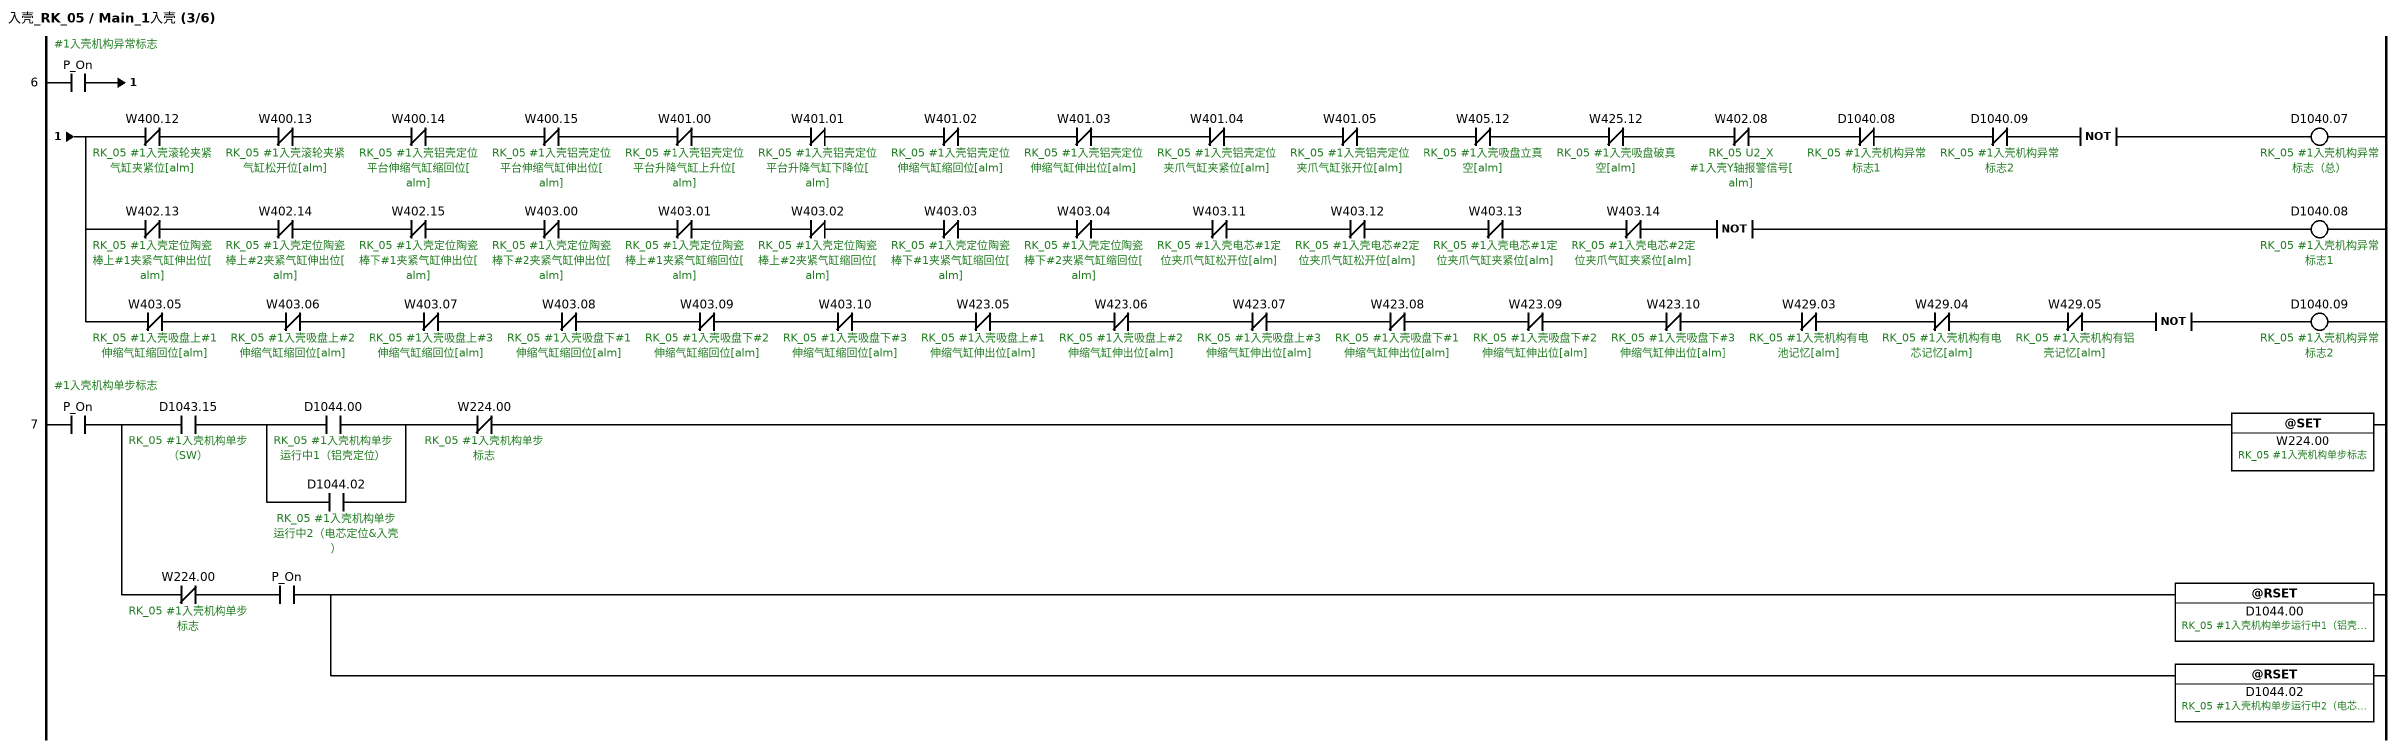
; [picture p408: 入壳_RK_05 / Main_1入壳, rungs 6-7]
; rung 6: #1入壳机构异常标志
LD P_On
OUT TR0
ANDNOT W400.12  ; RK_05 #1入壳滚轮夹紧气缸夹紧位[alm]
ANDNOT W400.13  ; RK_05 #1入壳滚轮夹紧气缸松开位[alm]
ANDNOT W400.14  ; RK_05 #1入壳铝壳定位平台伸缩气缸缩回位[alm]
ANDNOT W400.15  ; RK_05 #1入壳铝壳定位平台伸缩气缸伸出位[alm]
ANDNOT W401.00  ; RK_05 #1入壳铝壳定位平台升降气缸上升位[alm]
ANDNOT W401.01  ; RK_05 #1入壳铝壳定位平台升降气缸下降位[alm]
ANDNOT W401.02  ; RK_05 #1入壳铝壳定位伸缩气缸缩回位[alm]
ANDNOT W401.03  ; RK_05 #1入壳铝壳定位伸缩气缸伸出位[alm]
ANDNOT W401.04  ; RK_05 #1入壳铝壳定位夹爪气缸夹紧位[alm]
ANDNOT W401.05  ; RK_05 #1入壳铝壳定位夹爪气缸张开位[alm]
ANDNOT W405.12  ; RK_05 #1入壳吸盘立真空[alm]
ANDNOT W425.12  ; RK_05 #1入壳吸盘破真空[alm]
ANDNOT W402.08  ; RK_05 U2_X #1入壳Y轴报警信号[alm]
ANDNOT D1040.08  ; RK_05 #1入壳机构异常标志1
ANDNOT D1040.09  ; RK_05 #1入壳机构异常标志2
NOT(520)
OUT D1040.07  ; RK_05 #1入壳机构异常标志（总）
LD TR0
ANDNOT W402.13  ; RK_05 #1入壳定位陶瓷棒上#1夹紧气缸伸出位[alm]
ANDNOT W402.14  ; RK_05 #1入壳定位陶瓷棒上#2夹紧气缸伸出位[alm]
ANDNOT W402.15  ; RK_05 #1入壳定位陶瓷棒下#1夹紧气缸伸出位[alm]
ANDNOT W403.00  ; RK_05 #1入壳定位陶瓷棒下#2夹紧气缸伸出位[alm]
ANDNOT W403.01  ; RK_05 #1入壳定位陶瓷棒上#1夹紧气缸缩回位[alm]
ANDNOT W403.02  ; RK_05 #1入壳定位陶瓷棒上#2夹紧气缸缩回位[alm]
ANDNOT W403.03  ; RK_05 #1入壳定位陶瓷棒下#1夹紧气缸缩回位[alm]
ANDNOT W403.04  ; RK_05 #1入壳定位陶瓷棒下#2夹紧气缸缩回位[alm]
ANDNOT W403.11  ; RK_05 #1入壳电芯#1定位夹爪气缸松开位[alm]
ANDNOT W403.12  ; RK_05 #1入壳电芯#2定位夹爪气缸松开位[alm]
ANDNOT W403.13  ; RK_05 #1入壳电芯#1定位夹爪气缸夹紧位[alm]
ANDNOT W403.14  ; RK_05 #1入壳电芯#2定位夹爪气缸夹紧位[alm]
NOT(520)
OUT D1040.08  ; RK_05 #1入壳机构异常标志1
LD TR0
ANDNOT W403.05  ; RK_05 #1入壳吸盘上#1伸缩气缸缩回位[alm]
ANDNOT W403.06  ; RK_05 #1入壳吸盘上#2伸缩气缸缩回位[alm]
ANDNOT W403.07  ; RK_05 #1入壳吸盘上#3伸缩气缸缩回位[alm]
ANDNOT W403.08  ; RK_05 #1入壳吸盘下#1伸缩气缸缩回位[alm]
ANDNOT W403.09  ; RK_05 #1入壳吸盘下#2伸缩气缸缩回位[alm]
ANDNOT W403.10  ; RK_05 #1入壳吸盘下#3伸缩气缸缩回位[alm]
ANDNOT W423.05  ; RK_05 #1入壳吸盘上#1伸缩气缸伸出位[alm]
ANDNOT W423.06  ; RK_05 #1入壳吸盘上#2伸缩气缸伸出位[alm]
ANDNOT W423.07  ; RK_05 #1入壳吸盘上#3伸缩气缸伸出位[alm]
ANDNOT W423.08  ; RK_05 #1入壳吸盘下#1伸缩气缸伸出位[alm]
ANDNOT W423.09  ; RK_05 #1入壳吸盘下#2伸缩气缸伸出位[alm]
ANDNOT W423.10  ; RK_05 #1入壳吸盘下#3伸缩气缸伸出位[alm]
ANDNOT W429.03  ; RK_05 #1入壳机构有电池记忆[alm]
ANDNOT W429.04  ; RK_05 #1入壳机构有电芯记忆[alm]
ANDNOT W429.05  ; RK_05 #1入壳机构有铝壳记忆[alm]
NOT(520)
OUT D1040.09  ; RK_05 #1入壳机构异常标志2
; rung 7: #1入壳机构单步标志
LD P_On
OUT TR0
AND D1043.15  ; RK_05 #1入壳机构单步（SW）
LD D1044.00  ; RK_05 #1入壳机构单步运行中1（铝壳定位）
OR D1044.02  ; RK_05 #1入壳机构单步运行中2（电芯定位&入壳）
ANDLD
ANDNOT W224.00  ; RK_05 #1入壳机构单步标志
@SET W224.00  ; RK_05 #1入壳机构单步标志
LD TR0
ANDNOT W224.00  ; RK_05 #1入壳机构单步标志
AND P_On
@RSET D1044.00  ; RK_05 #1入壳机构单步运行中1（铝壳定位）
@RSET D1044.02  ; RK_05 #1入壳机构单步运行中2（电芯定位&入壳）

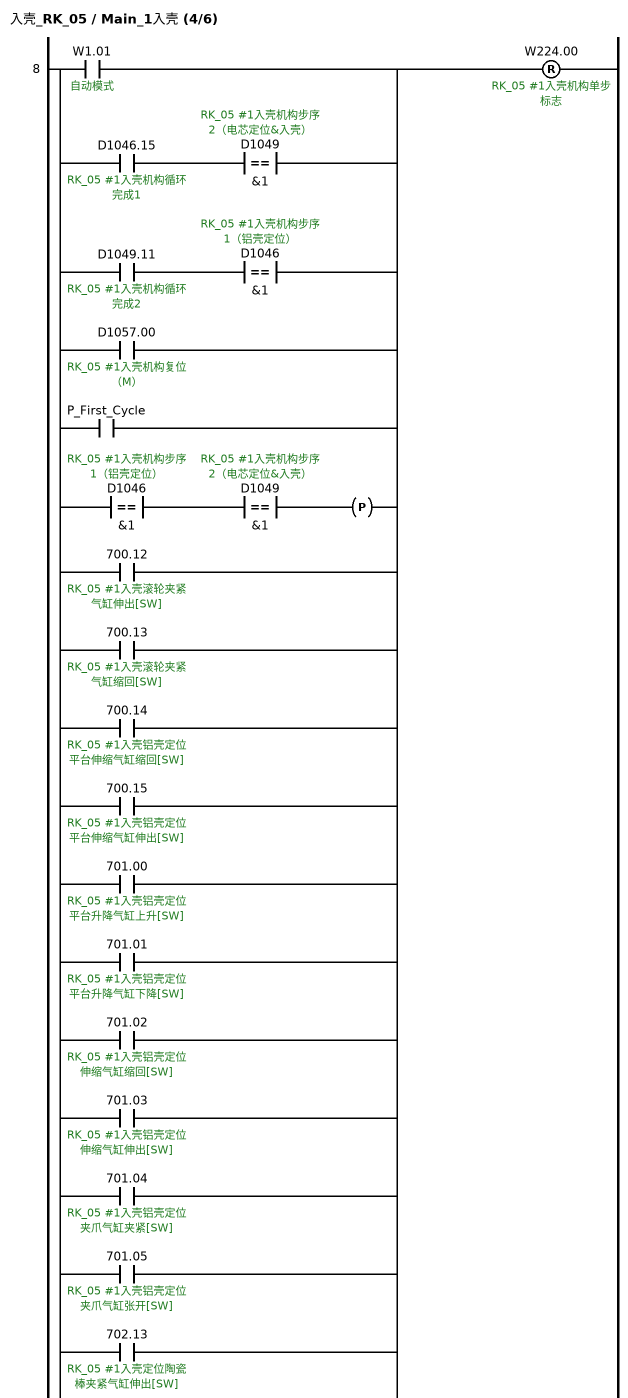

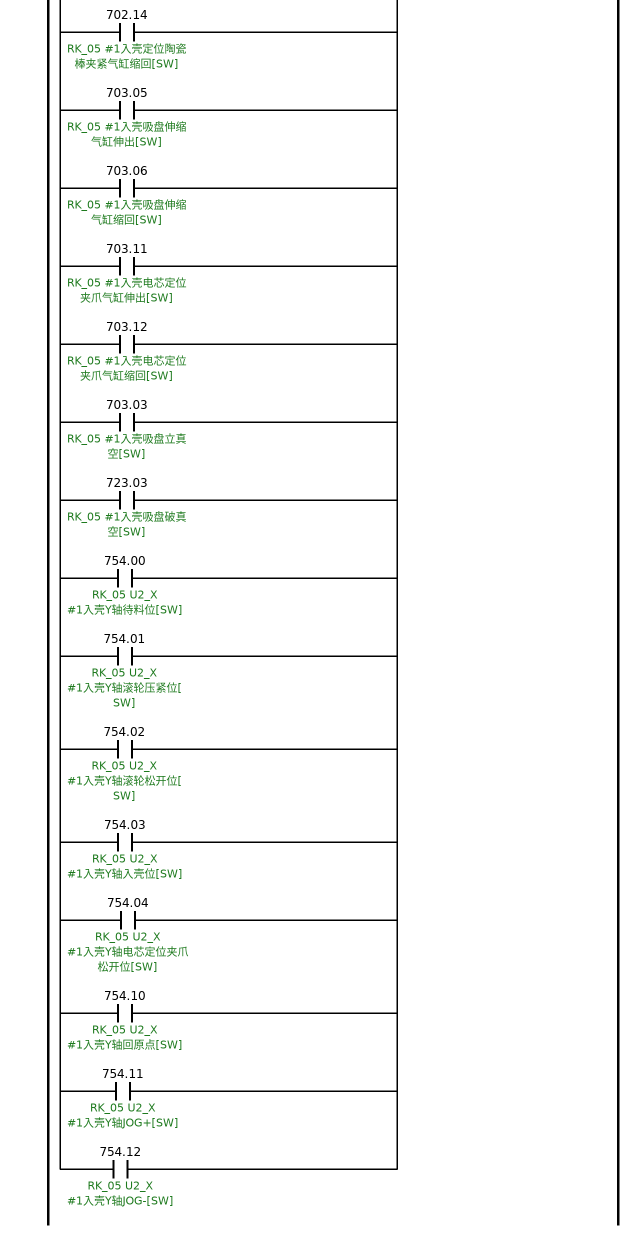
; rung 8
LD W1.01  ; 自动模式
LD D1046.15  ; RK_05 #1入壳机构循环完成1
AND=(300) D1049 &1  ; RK_05 #1入壳机构步序2（电芯定位&入壳）
ORLD
LD D1049.11  ; RK_05 #1入壳机构循环完成2
AND=(300) D1046 &1  ; RK_05 #1入壳机构步序1（铝壳定位）
ORLD
OR D1057.00  ; RK_05 #1入壳机构复位（M）
OR P_First_Cycle
LD=(300) D1046 &1  ; RK_05 #1入壳机构步序1（铝壳定位）
AND=(300) D1049 &1  ; RK_05 #1入壳机构步序2（电芯定位&入壳）
UP(521)
ORLD
OR 700.12  ; RK_05 #1入壳滚轮夹紧气缸伸出[SW]
OR 700.13  ; RK_05 #1入壳滚轮夹紧气缸缩回[SW]
OR 700.14  ; RK_05 #1入壳铝壳定位平台伸缩气缸缩回[SW]
OR 700.15  ; RK_05 #1入壳铝壳定位平台伸缩气缸伸出[SW]
OR 701.00  ; RK_05 #1入壳铝壳定位平台升降气缸上升[SW]
OR 701.01  ; RK_05 #1入壳铝壳定位平台升降气缸下降[SW]
OR 701.02  ; RK_05 #1入壳铝壳定位伸缩气缸缩回[SW]
OR 701.03  ; RK_05 #1入壳铝壳定位伸缩气缸伸出[SW]
OR 701.04  ; RK_05 #1入壳铝壳定位夹爪气缸夹紧[SW]
OR 701.05  ; RK_05 #1入壳铝壳定位夹爪气缸张开[SW]
OR 702.13  ; RK_05 #1入壳定位陶瓷棒夹紧气缸伸出[SW]
OR 702.14  ; RK_05 #1入壳定位陶瓷棒夹紧气缸缩回[SW]
OR 703.05  ; RK_05 #1入壳吸盘伸缩气缸伸出[SW]
OR 703.06  ; RK_05 #1入壳吸盘伸缩气缸缩回[SW]
OR 703.11  ; RK_05 #1入壳电芯定位夹爪气缸伸出[SW]
OR 703.12  ; RK_05 #1入壳电芯定位夹爪气缸缩回[SW]
OR 703.03  ; RK_05 #1入壳吸盘立真空[SW]
OR 723.03  ; RK_05 #1入壳吸盘破真空[SW]
OR 754.00  ; RK_05 U2_X #1入壳Y轴待料位[SW]
OR 754.01  ; RK_05 U2_X #1入壳Y轴滚轮压紧位[SW]
OR 754.02  ; RK_05 U2_X #1入壳Y轴滚轮松开位[SW]
OR 754.03  ; RK_05 U2_X #1入壳Y轴入壳位[SW]
OR 754.04  ; RK_05 U2_X #1入壳Y轴电芯定位夹爪松开位[SW]
OR 754.10  ; RK_05 U2_X #1入壳Y轴回原点[SW]
OR 754.11  ; RK_05 U2_X #1入壳Y轴JOG+[SW]
OR 754.12  ; RK_05 U2_X #1入壳Y轴JOG-[SW]
RSET W224.00  ; RK_05 #1入壳机构单步标志

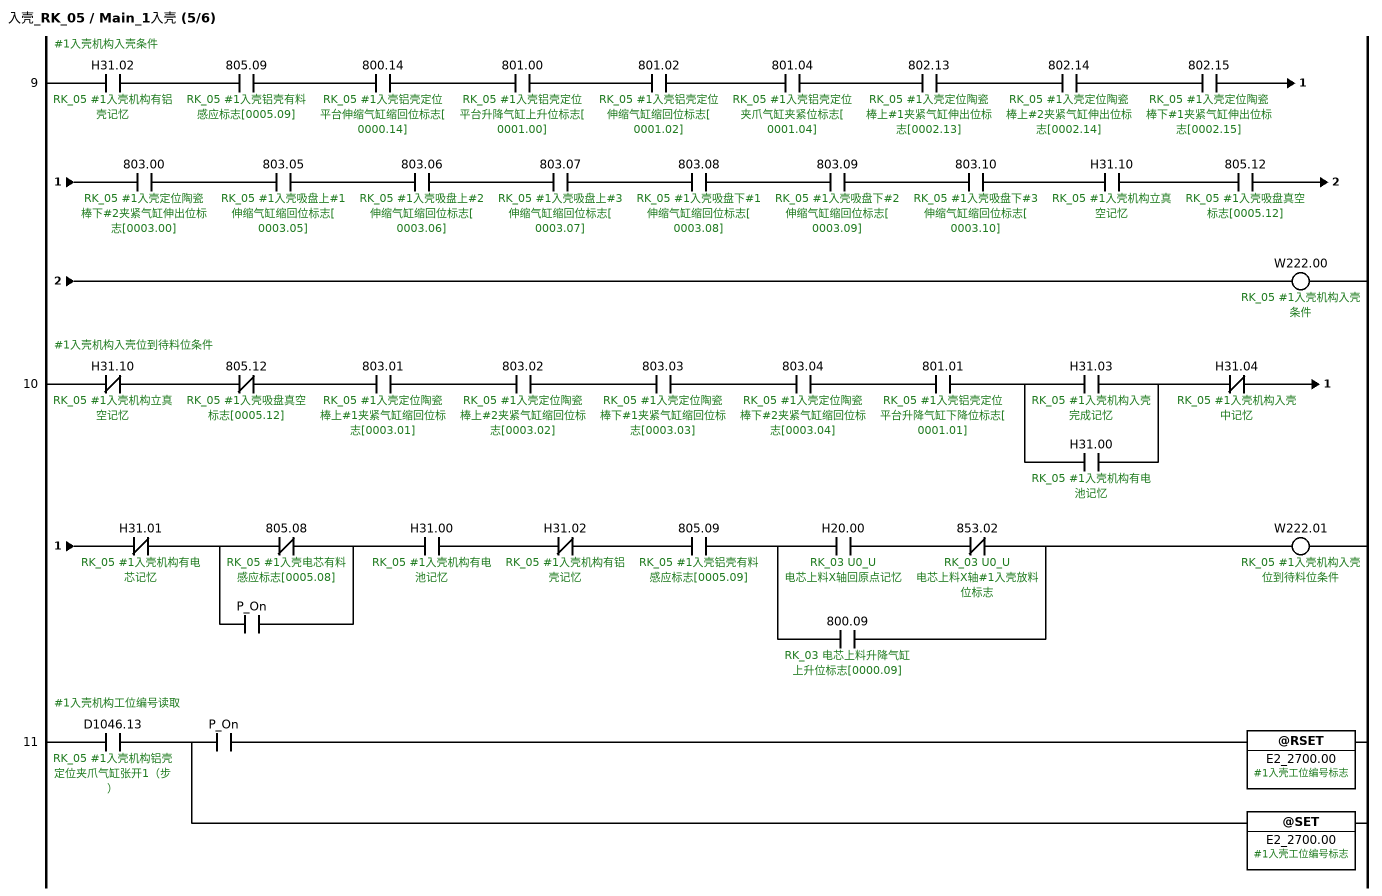
; rung 9: #1入壳机构入壳条件
LD H31.02  ; RK_05 #1入壳机构有铝壳记忆
AND 805.09  ; RK_05 #1入壳铝壳有料感应标志[0005.09]
AND 800.14  ; RK_05 #1入壳铝壳定位平台伸缩气缸缩回位标志[0000.14]
AND 801.00  ; RK_05 #1入壳铝壳定位平台升降气缸上升位标志[0001.00]
AND 801.02  ; RK_05 #1入壳铝壳定位伸缩气缸缩回位标志[0001.02]
AND 801.04  ; RK_05 #1入壳铝壳定位夹爪气缸夹紧位标志[0001.04]
AND 802.13  ; RK_05 #1入壳定位陶瓷棒上#1夹紧气缸伸出位标志[0002.13]
AND 802.14  ; RK_05 #1入壳定位陶瓷棒上#2夹紧气缸伸出位标志[0002.14]
AND 802.15  ; RK_05 #1入壳定位陶瓷棒下#1夹紧气缸伸出位标志[0002.15]
AND 803.00  ; RK_05 #1入壳定位陶瓷棒下#2夹紧气缸伸出位标志[0003.00]
AND 803.05  ; RK_05 #1入壳吸盘上#1伸缩气缸缩回位标志[0003.05]
AND 803.06  ; RK_05 #1入壳吸盘上#2伸缩气缸缩回位标志[0003.06]
AND 803.07  ; RK_05 #1入壳吸盘上#3伸缩气缸缩回位标志[0003.07]
AND 803.08  ; RK_05 #1入壳吸盘下#1伸缩气缸缩回位标志[0003.08]
AND 803.09  ; RK_05 #1入壳吸盘下#2伸缩气缸缩回位标志[0003.09]
AND 803.10  ; RK_05 #1入壳吸盘下#3伸缩气缸缩回位标志[0003.10]
AND H31.10  ; RK_05 #1入壳机构立真空记忆
AND 805.12  ; RK_05 #1入壳吸盘真空标志[0005.12]
OUT W222.00  ; RK_05 #1入壳机构入壳条件
; rung 10: #1入壳机构入壳位到待料位条件
LDNOT H31.10  ; RK_05 #1入壳机构立真空记忆
ANDNOT 805.12  ; RK_05 #1入壳吸盘真空标志[0005.12]
AND 803.01  ; RK_05 #1入壳定位陶瓷棒上#1夹紧气缸缩回位标志[0003.01]
AND 803.02  ; RK_05 #1入壳定位陶瓷棒上#2夹紧气缸缩回位标志[0003.02]
AND 803.03  ; RK_05 #1入壳定位陶瓷棒下#1夹紧气缸缩回位标志[0003.03]
AND 803.04  ; RK_05 #1入壳定位陶瓷棒下#2夹紧气缸缩回位标志[0003.04]
AND 801.01  ; RK_05 #1入壳铝壳定位平台升降气缸下降位标志[0001.01]
LD H31.03  ; RK_05 #1入壳机构入壳完成记忆
OR H31.00  ; RK_05 #1入壳机构有电池记忆
ANDLD
ANDNOT H31.04  ; RK_05 #1入壳机构入壳中记忆
ANDNOT H31.01  ; RK_05 #1入壳机构有电芯记忆
LDNOT 805.08  ; RK_05 #1入壳电芯有料感应标志[0005.08]
OR P_On
ANDLD
AND H31.00  ; RK_05 #1入壳机构有电池记忆
ANDNOT H31.02  ; RK_05 #1入壳机构有铝壳记忆
AND 805.09  ; RK_05 #1入壳铝壳有料感应标志[0005.09]
LD H20.00  ; RK_03 U0_U 电芯上料X轴回原点记忆
ANDNOT 853.02  ; RK_03 U0_U 电芯上料X轴#1入壳放料位标志
OR 800.09  ; RK_03 电芯上料升降气缸上升位标志[0000.09]
ANDLD
OUT W222.01  ; RK_05 #1入壳机构入壳位到待料位条件
; rung 11: #1入壳机构工位编号读取
LD D1046.13  ; RK_05 #1入壳机构铝壳定位夹爪气缸张开1（步）
OUT TR0
AND P_On
@RSET E2_2700.00  ; #1入壳工位编号标志
LD TR0
@SET E2_2700.00  ; #1入壳工位编号标志

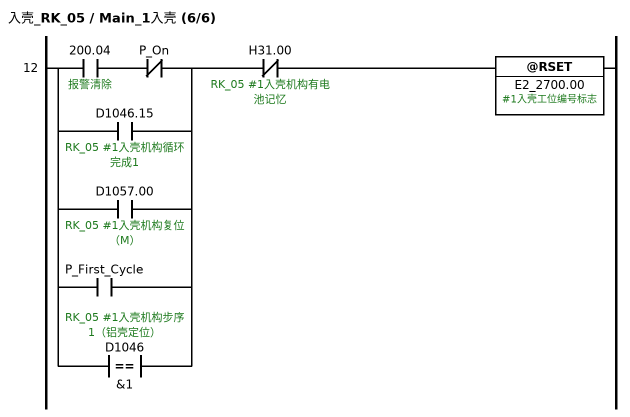
; rung 12
LD 200.04  ; 报警清除
ANDNOT P_On
OR D1046.15  ; RK_05 #1入壳机构循环完成1
OR D1057.00  ; RK_05 #1入壳机构复位（M）
OR P_First_Cycle
OR=(300) D1046 &1  ; RK_05 #1入壳机构步序1（铝壳定位）
ANDNOT H31.00  ; RK_05 #1入壳机构有电池记忆
@RSET E2_2700.00  ; #1入壳工位编号标志

### Section Main_2入壳

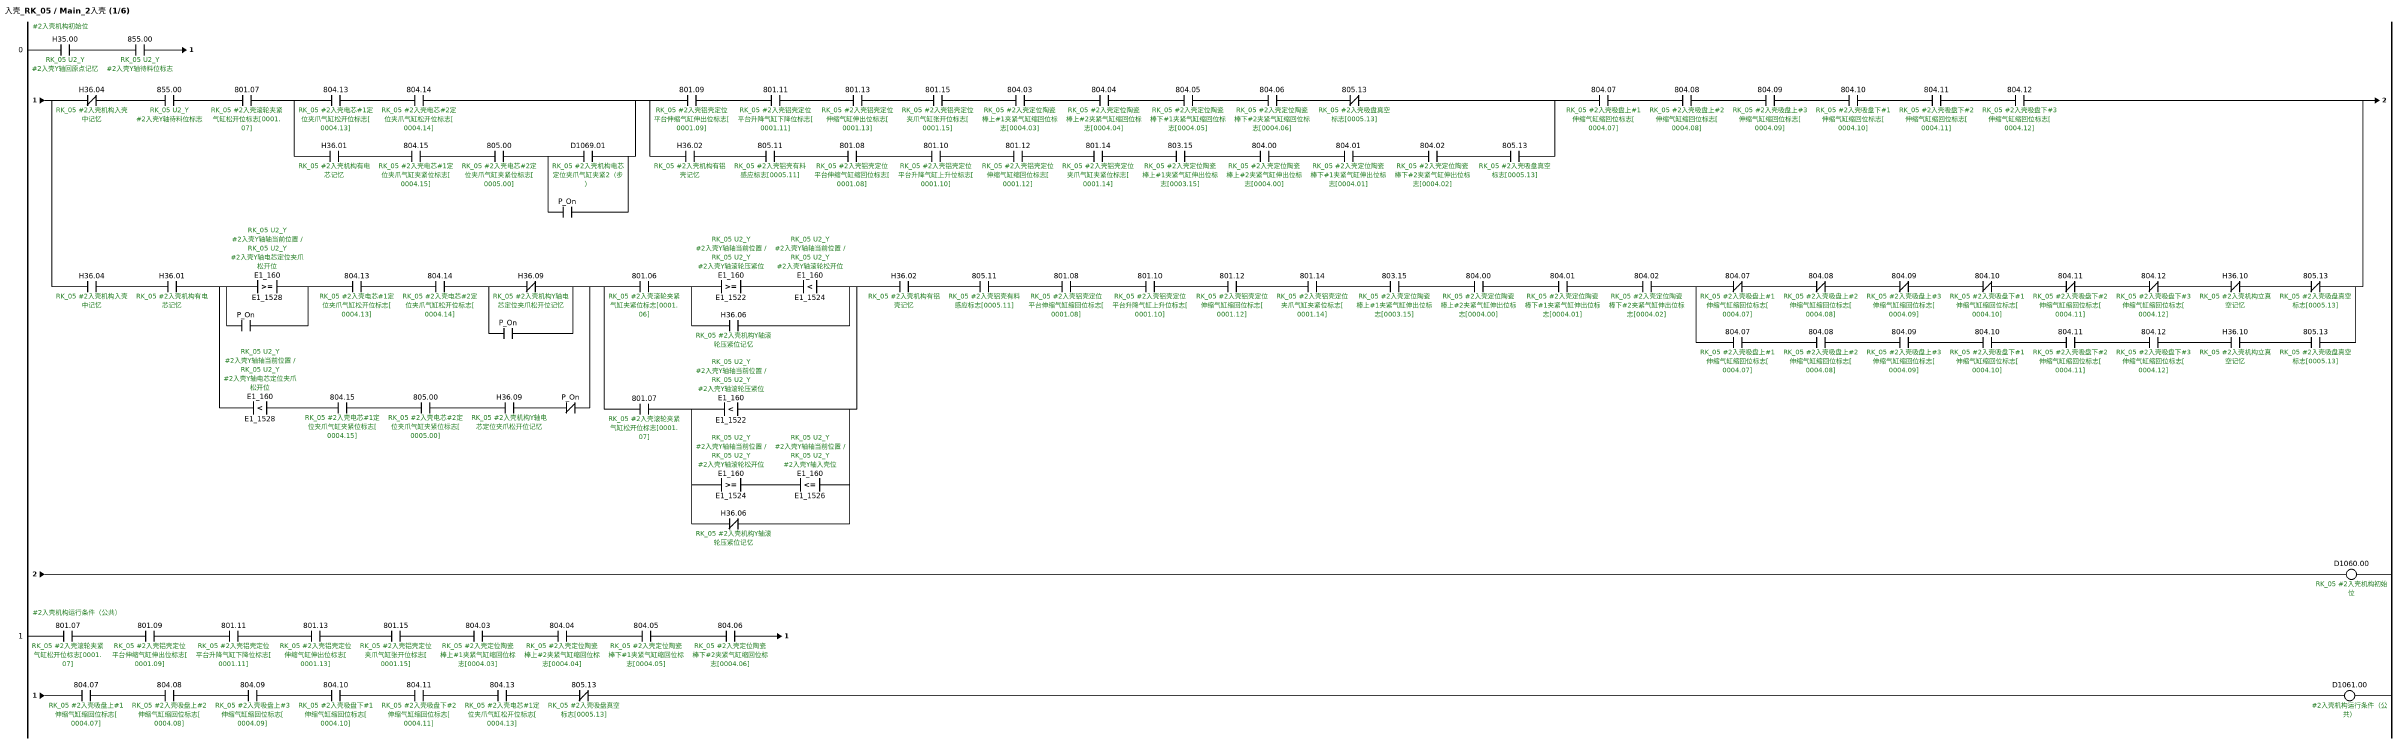
; rung 0: #2入壳机构初始位
LD H35.00  ; RK_05 U2_Y #2入壳Y轴回原点记忆
AND 855.00  ; RK_05 U2_Y #2入壳Y轴待料位标志
LDNOT H36.04  ; RK_05 #2入壳机构入壳中记忆
AND 855.00  ; RK_05 U2_Y #2入壳Y轴待料位标志
AND 801.07  ; RK_05 #2入壳滚轮夹紧气缸松开位标志[0001.07]
LD 804.13  ; RK_05 #2入壳电芯#1定位夹爪气缸松开位标志[0004.13]
AND 804.14  ; RK_05 #2入壳电芯#2定位夹爪气缸松开位标志[0004.14]
LD H36.01  ; RK_05 #2入壳机构有电芯记忆
AND 804.15  ; RK_05 #2入壳电芯#1定位夹爪气缸夹紧位标志[0004.15]
AND 805.00  ; RK_05 #2入壳电芯#2定位夹爪气缸夹紧位标志[0005.00]
LD D1069.01  ; RK_05 #2入壳机构电芯定位夹爪气缸夹紧2（步）
OR P_On
ANDLD
ORLD
ANDLD
LD 801.09  ; RK_05 #2入壳铝壳定位平台伸缩气缸伸出位标志[0001.09]
AND 801.11  ; RK_05 #2入壳铝壳定位平台升降气缸下降位标志[0001.11]
AND 801.13  ; RK_05 #2入壳铝壳定位伸缩气缸伸出位标志[0001.13]
AND 801.15  ; RK_05 #2入壳铝壳定位夹爪气缸张开位标志[0001.15]
AND 804.03  ; RK_05 #2入壳定位陶瓷棒上#1夹紧气缸缩回位标志[0004.03]
AND 804.04  ; RK_05 #2入壳定位陶瓷棒上#2夹紧气缸缩回位标志[0004.04]
AND 804.05  ; RK_05 #2入壳定位陶瓷棒下#1夹紧气缸缩回位标志[0004.05]
AND 804.06  ; RK_05 #2入壳定位陶瓷棒下#2夹紧气缸缩回位标志[0004.06]
ANDNOT 805.13  ; RK_05 #2入壳吸盘真空标志[0005.13]
LD H36.02  ; RK_05 #2入壳机构有铝壳记忆  // 20181014新增
AND 805.11  ; RK_05 #2入壳铝壳有料感应标志[0005.11]
AND 801.08  ; RK_05 #2入壳铝壳定位平台伸缩气缸缩回位标志[0001.08]
AND 801.10  ; RK_05 #2入壳铝壳定位平台升降气缸上升位标志[0001.10]
AND 801.12  ; RK_05 #2入壳铝壳定位伸缩气缸缩回位标志[0001.12]
AND 801.14  ; RK_05 #2入壳铝壳定位夹爪气缸夹紧位标志[0001.14]
AND 803.15  ; RK_05 #2入壳定位陶瓷棒上#1夹紧气缸伸出位标志[0003.15]
AND 804.00  ; RK_05 #2入壳定位陶瓷棒上#2夹紧气缸伸出位标志[0004.00]
AND 804.01  ; RK_05 #2入壳定位陶瓷棒下#1夹紧气缸伸出位标志[0004.01]
AND 804.02  ; RK_05 #2入壳定位陶瓷棒下#2夹紧气缸伸出位标志[0004.02]
AND 805.13  ; RK_05 #2入壳吸盘真空标志[0005.13]
ORLD
ANDLD
AND 804.07  ; RK_05 #2入壳吸盘上#1伸缩气缸缩回位标志[0004.07]
AND 804.08  ; RK_05 #2入壳吸盘上#2伸缩气缸缩回位标志[0004.08]
AND 804.09  ; RK_05 #2入壳吸盘上#3伸缩气缸缩回位标志[0004.09]
AND 804.10  ; RK_05 #2入壳吸盘下#1伸缩气缸缩回位标志[0004.10]
AND 804.11  ; RK_05 #2入壳吸盘下#2伸缩气缸缩回位标志[0004.11]
AND 804.12  ; RK_05 #2入壳吸盘下#3伸缩气缸缩回位标志[0004.12]
LD H36.04  ; RK_05 #2入壳机构入壳中记忆
AND H36.01  ; RK_05 #2入壳机构有电芯记忆
LD>=SL(328) E1_160 E1_1528  ; RK_05 U2_Y #2入壳Y轴轴当前位置, RK_05 U2_Y #2入壳Y轴电芯定位夹爪松开位
OR P_On
AND 804.13  ; RK_05 #2入壳电芯#1定位夹爪气缸松开位标志[0004.13]
AND 804.14  ; RK_05 #2入壳电芯#2定位夹爪气缸松开位标志[0004.14]
LDNOT H36.09  ; RK_05 #2入壳机构Y轴电芯定位夹爪松开位记忆
OR P_On
ANDLD
LD<SL(313) E1_160 E1_1528  ; RK_05 U2_Y #2入壳Y轴轴当前位置, RK_05 U2_Y #2入壳Y轴电芯定位夹爪松开位
AND 804.15  ; RK_05 #2入壳电芯#1定位夹爪气缸夹紧位标志[0004.15]
AND 805.00  ; RK_05 #2入壳电芯#2定位夹爪气缸夹紧位标志[0005.00]
AND H36.09  ; RK_05 #2入壳机构Y轴电芯定位夹爪松开位记忆
ANDNOT P_On
ORLD
ANDLD
LD 801.06  ; RK_05 #2入壳滚轮夹紧气缸夹紧位标志[0001.06]
LD>=SL(328) E1_160 E1_1522  ; RK_05 U2_Y #2入壳Y轴轴当前位置, RK_05 U2_Y #2入壳Y轴滚轮压紧位
AND<SL(313) E1_160 E1_1524  ; RK_05 U2_Y #2入壳Y轴轴当前位置, RK_05 U2_Y #2入壳Y轴滚轮松开位
OR H36.06  ; RK_05 #2入壳机构Y轴滚轮压紧位记忆
ANDLD
LD 801.07  ; RK_05 #2入壳滚轮夹紧气缸松开位标志[0001.07]
LD<SL(313) E1_160 E1_1522  ; RK_05 U2_Y #2入壳Y轴轴当前位置, RK_05 U2_Y #2入壳Y轴滚轮压紧位
LD>=SL(328) E1_160 E1_1524  ; RK_05 U2_Y #2入壳Y轴轴当前位置, RK_05 U2_Y #2入壳Y轴滚轮松开位
AND<=SL(318) E1_160 E1_1526  ; RK_05 U2_Y #2入壳Y轴轴当前位置, RK_05 U2_Y #2入壳Y轴入壳位
ORLD
ORNOT H36.06  ; RK_05 #2入壳机构Y轴滚轮压紧位记忆
ANDLD
ORLD
ANDLD
AND H36.02  ; RK_05 #2入壳机构有铝壳记忆
AND 805.11  ; RK_05 #2入壳铝壳有料感应标志[0005.11]
AND 801.08  ; RK_05 #2入壳铝壳定位平台伸缩气缸缩回位标志[0001.08]
AND 801.10  ; RK_05 #2入壳铝壳定位平台升降气缸上升位标志[0001.10]
AND 801.12  ; RK_05 #2入壳铝壳定位伸缩气缸缩回位标志[0001.12]
AND 801.14  ; RK_05 #2入壳铝壳定位夹爪气缸夹紧位标志[0001.14]
AND 803.15  ; RK_05 #2入壳定位陶瓷棒上#1夹紧气缸伸出位标志[0003.15]
AND 804.00  ; RK_05 #2入壳定位陶瓷棒上#2夹紧气缸伸出位标志[0004.00]
AND 804.01  ; RK_05 #2入壳定位陶瓷棒下#1夹紧气缸伸出位标志[0004.01]
AND 804.02  ; RK_05 #2入壳定位陶瓷棒下#2夹紧气缸伸出位标志[0004.02]
LDNOT 804.07  ; RK_05 #2入壳吸盘上#1伸缩气缸缩回位标志[0004.07]
ANDNOT 804.08  ; RK_05 #2入壳吸盘上#2伸缩气缸缩回位标志[0004.08]
ANDNOT 804.09  ; RK_05 #2入壳吸盘上#3伸缩气缸缩回位标志[0004.09]
ANDNOT 804.10  ; RK_05 #2入壳吸盘下#1伸缩气缸缩回位标志[0004.10]
ANDNOT 804.11  ; RK_05 #2入壳吸盘下#2伸缩气缸缩回位标志[0004.11]
ANDNOT 804.12  ; RK_05 #2入壳吸盘下#3伸缩气缸缩回位标志[0004.12]
ANDNOT H36.10  ; RK_05 #2入壳机构立真空记忆
ANDNOT 805.13  ; RK_05 #2入壳吸盘真空标志[0005.13]
LD 804.07  ; RK_05 #2入壳吸盘上#1伸缩气缸缩回位标志[0004.07]
AND 804.08  ; RK_05 #2入壳吸盘上#2伸缩气缸缩回位标志[0004.08]
AND 804.09  ; RK_05 #2入壳吸盘上#3伸缩气缸缩回位标志[0004.09]
AND 804.10  ; RK_05 #2入壳吸盘下#1伸缩气缸缩回位标志[0004.10]
AND 804.11  ; RK_05 #2入壳吸盘下#2伸缩气缸缩回位标志[0004.11]
AND 804.12  ; RK_05 #2入壳吸盘下#3伸缩气缸缩回位标志[0004.12]
AND H36.10  ; RK_05 #2入壳机构立真空记忆
AND 805.13  ; RK_05 #2入壳吸盘真空标志[0005.13]
ORLD
ANDLD
ORLD
ANDLD
OUT D1060.00  ; RK_05 #2入壳机构初始位
; rung 1: #2入壳机构运行条件（公共）
LD 801.07  ; RK_05 #2入壳滚轮夹紧气缸松开位标志[0001.07]
AND 801.09  ; RK_05 #2入壳铝壳定位平台伸缩气缸伸出位标志[0001.09]
AND 801.11  ; RK_05 #2入壳铝壳定位平台升降气缸下降位标志[0001.11]
AND 801.13  ; RK_05 #2入壳铝壳定位伸缩气缸伸出位标志[0001.13]
AND 801.15  ; RK_05 #2入壳铝壳定位夹爪气缸张开位标志[0001.15]
AND 804.03  ; RK_05 #2入壳定位陶瓷棒上#1夹紧气缸缩回位标志[0004.03]
AND 804.04  ; RK_05 #2入壳定位陶瓷棒上#2夹紧气缸缩回位标志[0004.04]
AND 804.05  ; RK_05 #2入壳定位陶瓷棒下#1夹紧气缸缩回位标志[0004.05]
AND 804.06  ; RK_05 #2入壳定位陶瓷棒下#2夹紧气缸缩回位标志[0004.06]
AND 804.07  ; RK_05 #2入壳吸盘上#1伸缩气缸缩回位标志[0004.07]
AND 804.08  ; RK_05 #2入壳吸盘上#2伸缩气缸缩回位标志[0004.08]
AND 804.09  ; RK_05 #2入壳吸盘上#3伸缩气缸缩回位标志[0004.09]
AND 804.10  ; RK_05 #2入壳吸盘下#1伸缩气缸缩回位标志[0004.10]
AND 804.11  ; RK_05 #2入壳吸盘下#2伸缩气缸缩回位标志[0004.11]
AND 804.13  ; RK_05 #2入壳电芯#1定位夹爪气缸松开位标志[0004.13]
ANDNOT 805.13  ; RK_05 #2入壳吸盘真空标志[0005.13]
OUT D1061.00  ; #2入壳机构运行条件（公共）

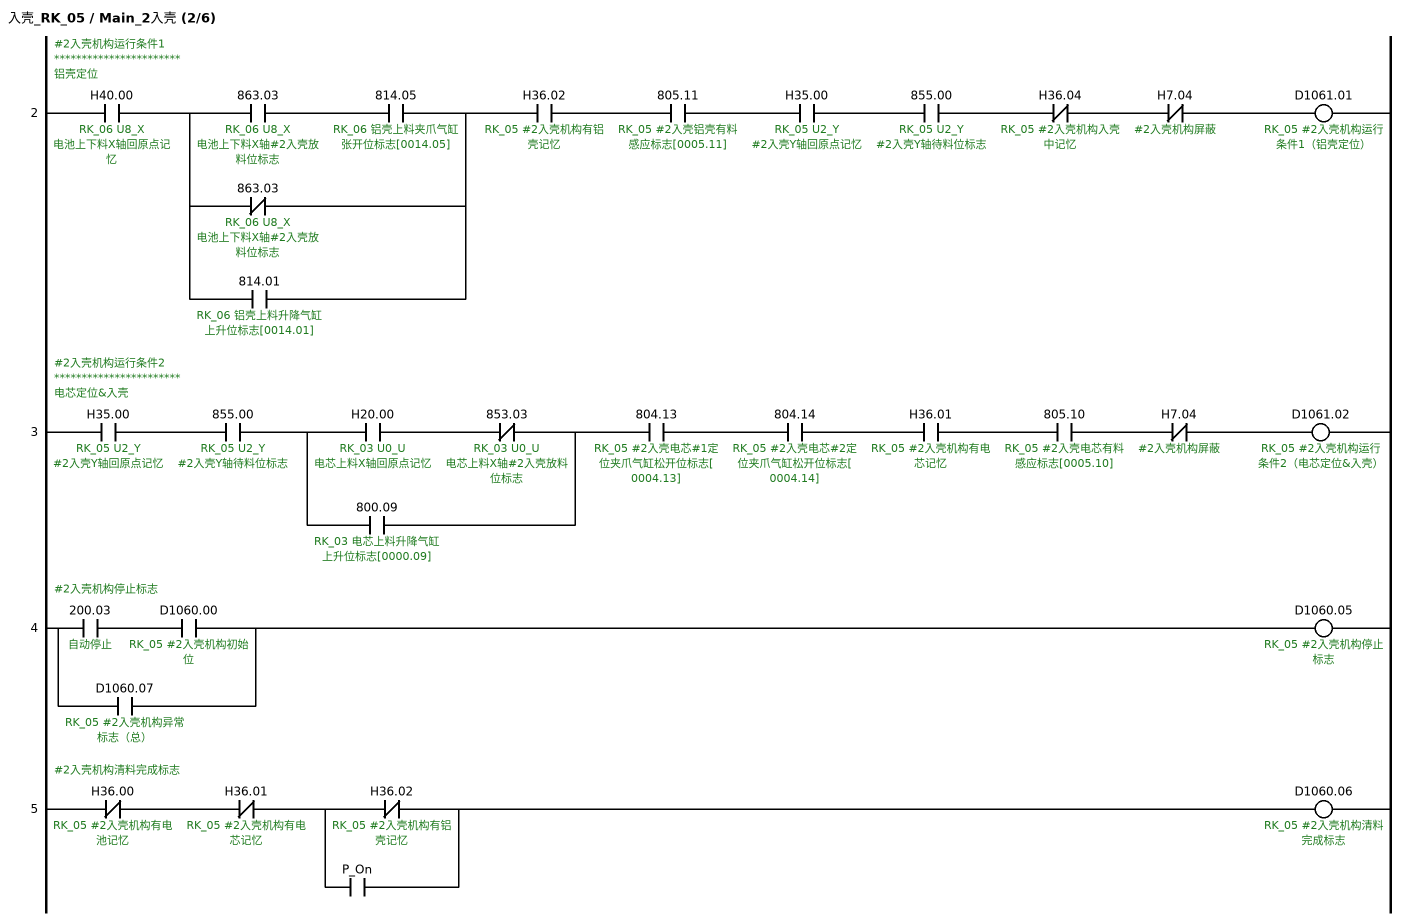
; rung 2: #2入壳机构运行条件1 / *********************** / 铝壳定位
LD H40.00  ; RK_06 U8_X 电池上下料X轴回原点记忆
LD 863.03  ; RK_06 U8_X 电池上下料X轴#2入壳放料位标志
AND 814.05  ; RK_06 铝壳上料夹爪气缸张开位标志[0014.05]
ORNOT 863.03  ; RK_06 U8_X 电池上下料X轴#2入壳放料位标志
OR 814.01  ; RK_06 铝壳上料升降气缸上升位标志[0014.01]
ANDLD
AND H36.02  ; RK_05 #2入壳机构有铝壳记忆
AND 805.11  ; RK_05 #2入壳铝壳有料感应标志[0005.11]
AND H35.00  ; RK_05 U2_Y #2入壳Y轴回原点记忆
AND 855.00  ; RK_05 U2_Y #2入壳Y轴待料位标志
ANDNOT H36.04  ; RK_05 #2入壳机构入壳中记忆
ANDNOT H7.04  ; #2入壳机构屏蔽
OUT D1061.01  ; RK_05 #2入壳机构运行条件1（铝壳定位）
; rung 3: #2入壳机构运行条件2 / *********************** / 电芯定位&入壳
LD H35.00  ; RK_05 U2_Y #2入壳Y轴回原点记忆
AND 855.00  ; RK_05 U2_Y #2入壳Y轴待料位标志
LD H20.00  ; RK_03 U0_U 电芯上料X轴回原点记忆
ANDNOT 853.03  ; RK_03 U0_U 电芯上料X轴#2入壳放料位标志
OR 800.09  ; RK_03 电芯上料升降气缸上升位标志[0000.09]
ANDLD
AND 804.13  ; RK_05 #2入壳电芯#1定位夹爪气缸松开位标志[0004.13]
AND 804.14  ; RK_05 #2入壳电芯#2定位夹爪气缸松开位标志[0004.14]
AND H36.01  ; RK_05 #2入壳机构有电芯记忆
AND 805.10  ; RK_05 #2入壳电芯有料感应标志[0005.10]
ANDNOT H7.04  ; #2入壳机构屏蔽
OUT D1061.02  ; RK_05 #2入壳机构运行条件2（电芯定位&入壳）
; rung 4: #2入壳机构停止标志
LD 200.03  ; 自动停止
AND D1060.00  ; RK_05 #2入壳机构初始位
OR D1060.07  ; RK_05 #2入壳机构异常标志（总）
OUT D1060.05  ; RK_05 #2入壳机构停止标志
; rung 5: #2入壳机构清料完成标志
LDNOT H36.00  ; RK_05 #2入壳机构有电池记忆
ANDNOT H36.01  ; RK_05 #2入壳机构有电芯记忆
LDNOT H36.02  ; RK_05 #2入壳机构有铝壳记忆
OR P_On
ANDLD
OUT D1060.06  ; RK_05 #2入壳机构清料完成标志

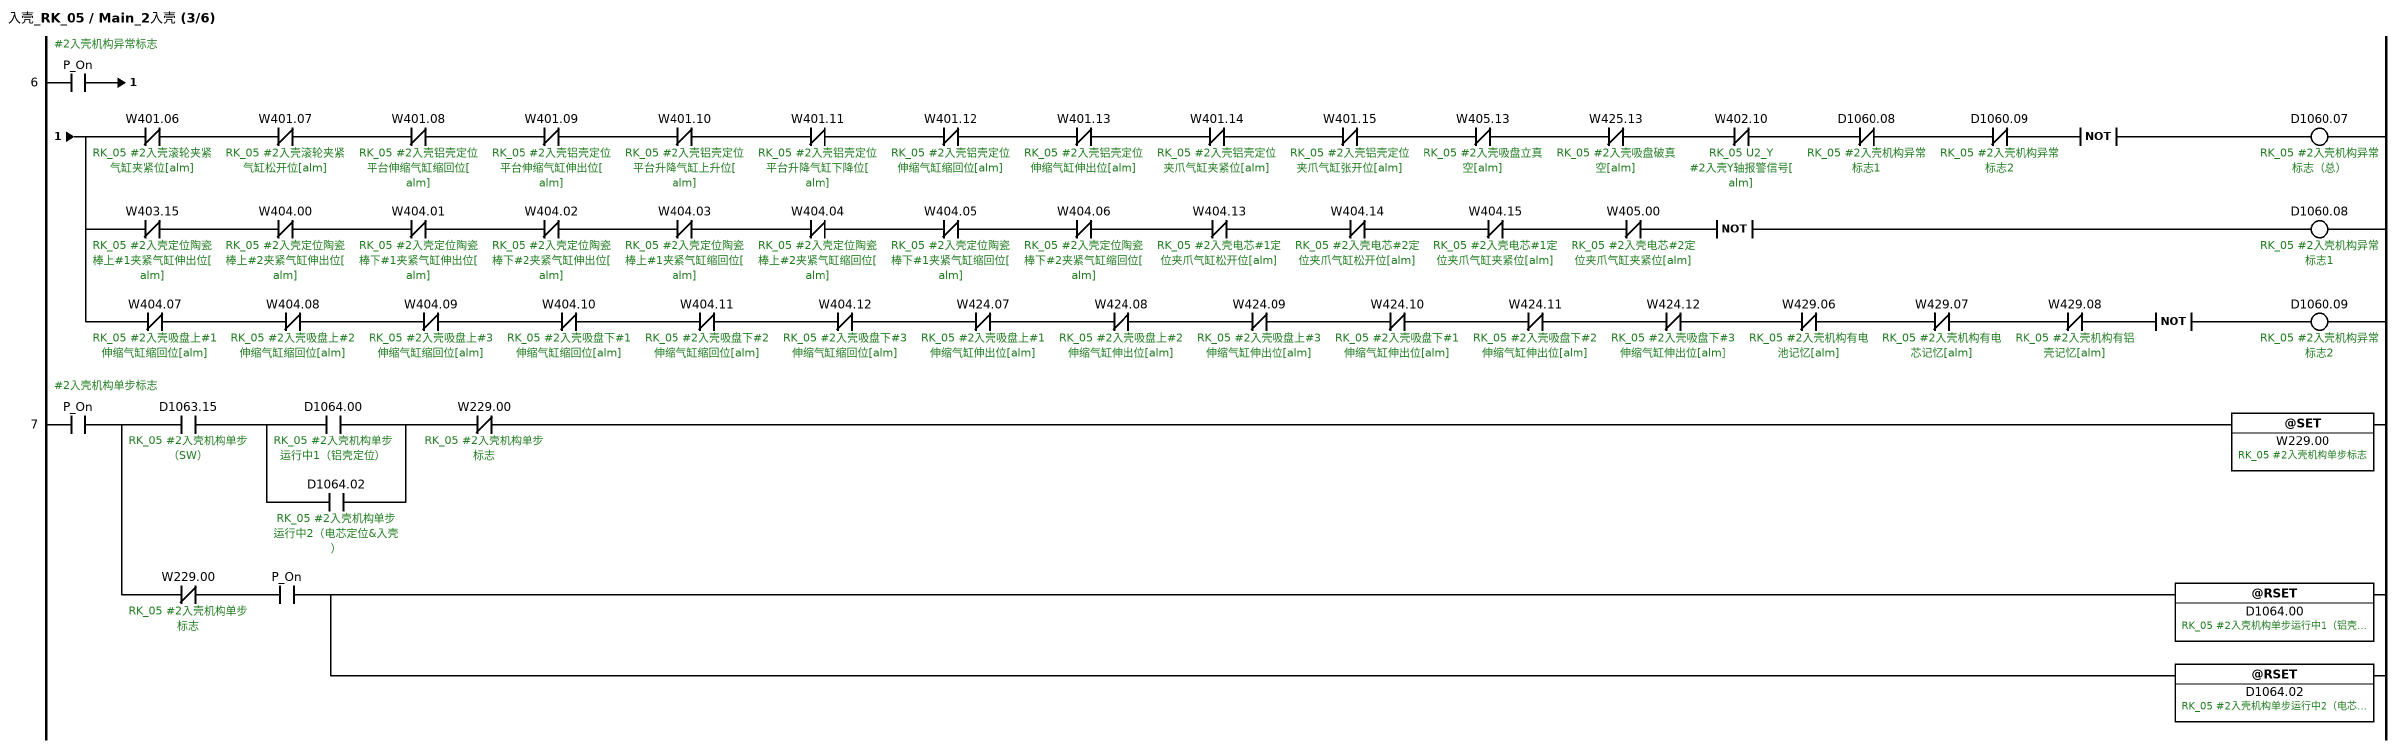
; rung 6: #2入壳机构异常标志
LD P_On
OUT TR0
ANDNOT W401.06  ; RK_05 #2入壳滚轮夹紧气缸夹紧位[alm]
ANDNOT W401.07  ; RK_05 #2入壳滚轮夹紧气缸松开位[alm]
ANDNOT W401.08  ; RK_05 #2入壳铝壳定位平台伸缩气缸缩回位[alm]
ANDNOT W401.09  ; RK_05 #2入壳铝壳定位平台伸缩气缸伸出位[alm]
ANDNOT W401.10  ; RK_05 #2入壳铝壳定位平台升降气缸上升位[alm]
ANDNOT W401.11  ; RK_05 #2入壳铝壳定位平台升降气缸下降位[alm]
ANDNOT W401.12  ; RK_05 #2入壳铝壳定位伸缩气缸缩回位[alm]
ANDNOT W401.13  ; RK_05 #2入壳铝壳定位伸缩气缸伸出位[alm]
ANDNOT W401.14  ; RK_05 #2入壳铝壳定位夹爪气缸夹紧位[alm]
ANDNOT W401.15  ; RK_05 #2入壳铝壳定位夹爪气缸张开位[alm]
ANDNOT W405.13  ; RK_05 #2入壳吸盘立真空[alm]
ANDNOT W425.13  ; RK_05 #2入壳吸盘破真空[alm]
ANDNOT W402.10  ; RK_05 U2_Y #2入壳Y轴报警信号[alm]
ANDNOT D1060.08  ; RK_05 #2入壳机构异常标志1
ANDNOT D1060.09  ; RK_05 #2入壳机构异常标志2
NOT(520)
OUT D1060.07  ; RK_05 #2入壳机构异常标志（总）
LD TR0
ANDNOT W403.15  ; RK_05 #2入壳定位陶瓷棒上#1夹紧气缸伸出位[alm]
ANDNOT W404.00  ; RK_05 #2入壳定位陶瓷棒上#2夹紧气缸伸出位[alm]
ANDNOT W404.01  ; RK_05 #2入壳定位陶瓷棒下#1夹紧气缸伸出位[alm]
ANDNOT W404.02  ; RK_05 #2入壳定位陶瓷棒下#2夹紧气缸伸出位[alm]
ANDNOT W404.03  ; RK_05 #2入壳定位陶瓷棒上#1夹紧气缸缩回位[alm]
ANDNOT W404.04  ; RK_05 #2入壳定位陶瓷棒上#2夹紧气缸缩回位[alm]
ANDNOT W404.05  ; RK_05 #2入壳定位陶瓷棒下#1夹紧气缸缩回位[alm]
ANDNOT W404.06  ; RK_05 #2入壳定位陶瓷棒下#2夹紧气缸缩回位[alm]
ANDNOT W404.13  ; RK_05 #2入壳电芯#1定位夹爪气缸松开位[alm]
ANDNOT W404.14  ; RK_05 #2入壳电芯#2定位夹爪气缸松开位[alm]
ANDNOT W404.15  ; RK_05 #2入壳电芯#1定位夹爪气缸夹紧位[alm]
ANDNOT W405.00  ; RK_05 #2入壳电芯#2定位夹爪气缸夹紧位[alm]
NOT(520)
OUT D1060.08  ; RK_05 #2入壳机构异常标志1
LD TR0
ANDNOT W404.07  ; RK_05 #2入壳吸盘上#1伸缩气缸缩回位[alm]
ANDNOT W404.08  ; RK_05 #2入壳吸盘上#2伸缩气缸缩回位[alm]
ANDNOT W404.09  ; RK_05 #2入壳吸盘上#3伸缩气缸缩回位[alm]
ANDNOT W404.10  ; RK_05 #2入壳吸盘下#1伸缩气缸缩回位[alm]
ANDNOT W404.11  ; RK_05 #2入壳吸盘下#2伸缩气缸缩回位[alm]
ANDNOT W404.12  ; RK_05 #2入壳吸盘下#3伸缩气缸缩回位[alm]
ANDNOT W424.07  ; RK_05 #2入壳吸盘上#1伸缩气缸伸出位[alm]
ANDNOT W424.08  ; RK_05 #2入壳吸盘上#2伸缩气缸伸出位[alm]
ANDNOT W424.09  ; RK_05 #2入壳吸盘上#3伸缩气缸伸出位[alm]
ANDNOT W424.10  ; RK_05 #2入壳吸盘下#1伸缩气缸伸出位[alm]
ANDNOT W424.11  ; RK_05 #2入壳吸盘下#2伸缩气缸伸出位[alm]
ANDNOT W424.12  ; RK_05 #2入壳吸盘下#3伸缩气缸伸出位[alm]
ANDNOT W429.06  ; RK_05 #2入壳机构有电池记忆[alm]
ANDNOT W429.07  ; RK_05 #2入壳机构有电芯记忆[alm]
ANDNOT W429.08  ; RK_05 #2入壳机构有铝壳记忆[alm]
NOT(520)
OUT D1060.09  ; RK_05 #2入壳机构异常标志2
; rung 7: #2入壳机构单步标志
LD P_On
OUT TR0
AND D1063.15  ; RK_05 #2入壳机构单步（SW）
LD D1064.00  ; RK_05 #2入壳机构单步运行中1（铝壳定位）
OR D1064.02  ; RK_05 #2入壳机构单步运行中2（电芯定位&入壳）
ANDLD
ANDNOT W229.00  ; RK_05 #2入壳机构单步标志
@SET W229.00  ; RK_05 #2入壳机构单步标志
LD TR0
ANDNOT W229.00  ; RK_05 #2入壳机构单步标志
AND P_On
@RSET D1064.00  ; RK_05 #2入壳机构单步运行中1（铝壳定位）
@RSET D1064.02  ; RK_05 #2入壳机构单步运行中2（电芯定位&入壳）

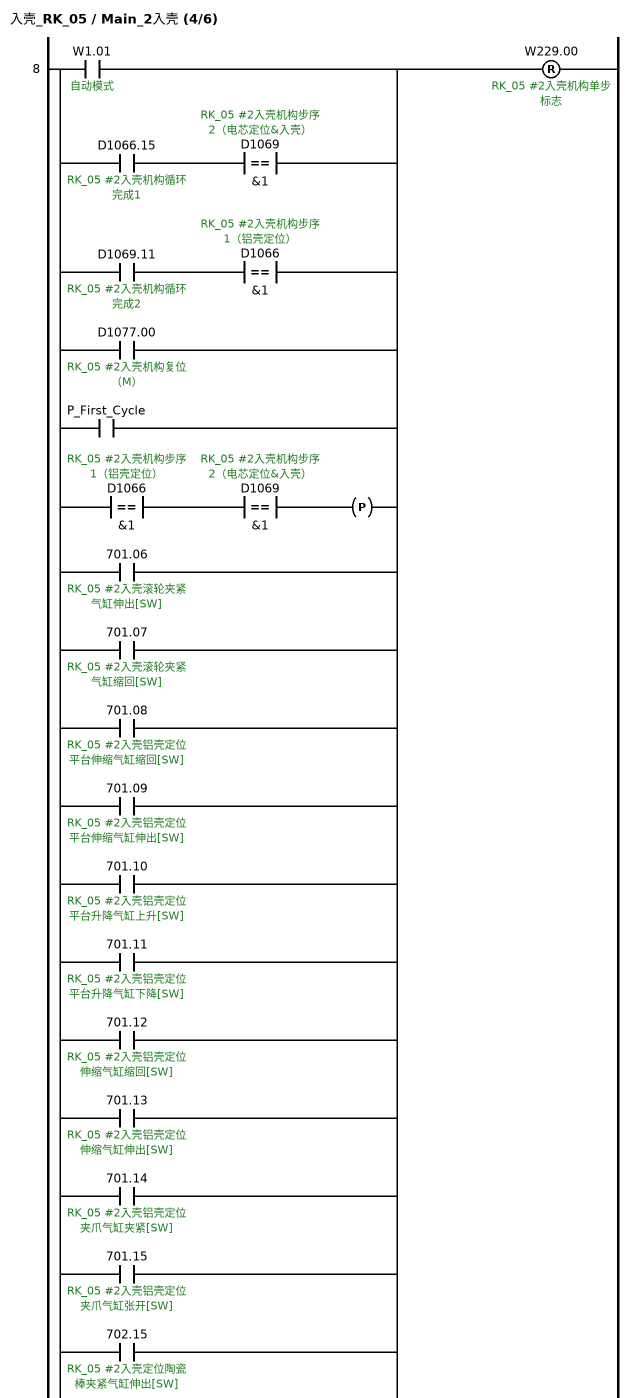

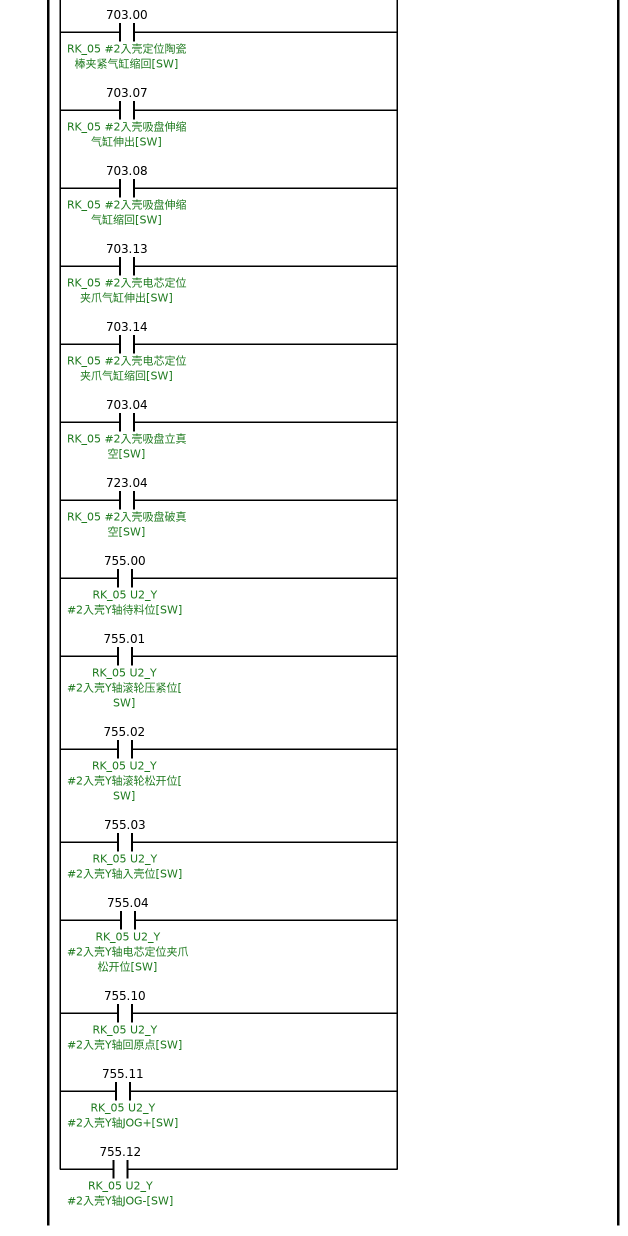
; rung 8
LD W1.01  ; 自动模式
LD D1066.15  ; RK_05 #2入壳机构循环完成1
AND=(300) D1069 &1  ; RK_05 #2入壳机构步序2（电芯定位&入壳）
ORLD
LD D1069.11  ; RK_05 #2入壳机构循环完成2
AND=(300) D1066 &1  ; RK_05 #2入壳机构步序1（铝壳定位）
ORLD
OR D1077.00  ; RK_05 #2入壳机构复位（M）
OR P_First_Cycle
LD=(300) D1066 &1  ; RK_05 #2入壳机构步序1（铝壳定位）
AND=(300) D1069 &1  ; RK_05 #2入壳机构步序2（电芯定位&入壳）
UP(521)
ORLD
OR 701.06  ; RK_05 #2入壳滚轮夹紧气缸伸出[SW]
OR 701.07  ; RK_05 #2入壳滚轮夹紧气缸缩回[SW]
OR 701.08  ; RK_05 #2入壳铝壳定位平台伸缩气缸缩回[SW]
OR 701.09  ; RK_05 #2入壳铝壳定位平台伸缩气缸伸出[SW]
OR 701.10  ; RK_05 #2入壳铝壳定位平台升降气缸上升[SW]
OR 701.11  ; RK_05 #2入壳铝壳定位平台升降气缸下降[SW]
OR 701.12  ; RK_05 #2入壳铝壳定位伸缩气缸缩回[SW]
OR 701.13  ; RK_05 #2入壳铝壳定位伸缩气缸伸出[SW]
OR 701.14  ; RK_05 #2入壳铝壳定位夹爪气缸夹紧[SW]
OR 701.15  ; RK_05 #2入壳铝壳定位夹爪气缸张开[SW]
OR 702.15  ; RK_05 #2入壳定位陶瓷棒夹紧气缸伸出[SW]
OR 703.00  ; RK_05 #2入壳定位陶瓷棒夹紧气缸缩回[SW]
OR 703.07  ; RK_05 #2入壳吸盘伸缩气缸伸出[SW]
OR 703.08  ; RK_05 #2入壳吸盘伸缩气缸缩回[SW]
OR 703.13  ; RK_05 #2入壳电芯定位夹爪气缸伸出[SW]
OR 703.14  ; RK_05 #2入壳电芯定位夹爪气缸缩回[SW]
OR 703.04  ; RK_05 #2入壳吸盘立真空[SW]
OR 723.04  ; RK_05 #2入壳吸盘破真空[SW]
OR 755.00  ; RK_05 U2_Y #2入壳Y轴待料位[SW]
OR 755.01  ; RK_05 U2_Y #2入壳Y轴滚轮压紧位[SW]
OR 755.02  ; RK_05 U2_Y #2入壳Y轴滚轮松开位[SW]
OR 755.03  ; RK_05 U2_Y #2入壳Y轴入壳位[SW]
OR 755.04  ; RK_05 U2_Y #2入壳Y轴电芯定位夹爪松开位[SW]
OR 755.10  ; RK_05 U2_Y #2入壳Y轴回原点[SW]
OR 755.11  ; RK_05 U2_Y #2入壳Y轴JOG+[SW]
OR 755.12  ; RK_05 U2_Y #2入壳Y轴JOG-[SW]
RSET W229.00  ; RK_05 #2入壳机构单步标志

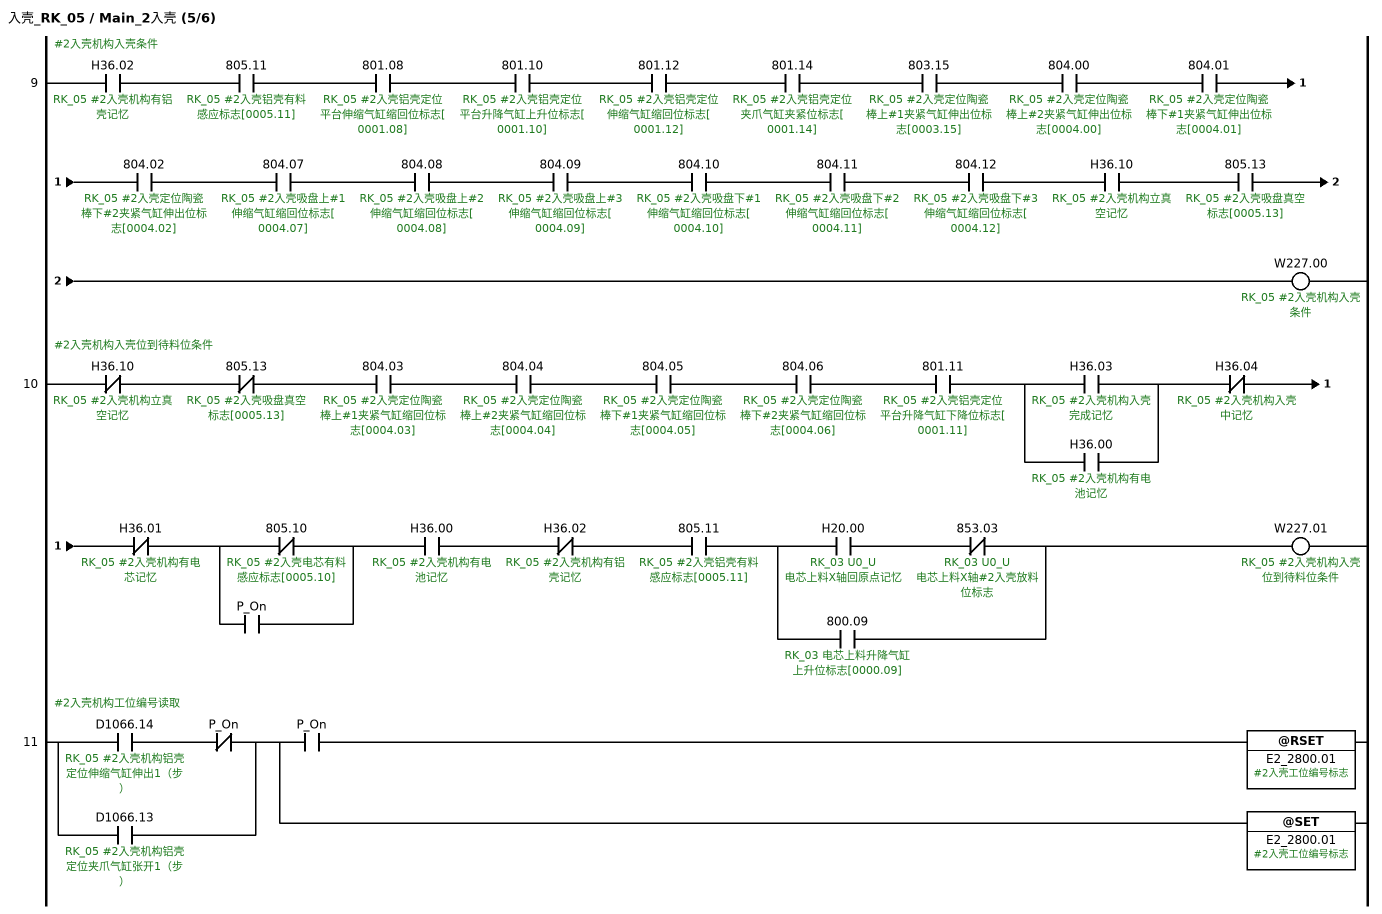
; rung 9: #2入壳机构入壳条件
LD H36.02  ; RK_05 #2入壳机构有铝壳记忆
AND 805.11  ; RK_05 #2入壳铝壳有料感应标志[0005.11]
AND 801.08  ; RK_05 #2入壳铝壳定位平台伸缩气缸缩回位标志[0001.08]
AND 801.10  ; RK_05 #2入壳铝壳定位平台升降气缸上升位标志[0001.10]
AND 801.12  ; RK_05 #2入壳铝壳定位伸缩气缸缩回位标志[0001.12]
AND 801.14  ; RK_05 #2入壳铝壳定位夹爪气缸夹紧位标志[0001.14]
AND 803.15  ; RK_05 #2入壳定位陶瓷棒上#1夹紧气缸伸出位标志[0003.15]
AND 804.00  ; RK_05 #2入壳定位陶瓷棒上#2夹紧气缸伸出位标志[0004.00]
AND 804.01  ; RK_05 #2入壳定位陶瓷棒下#1夹紧气缸伸出位标志[0004.01]
AND 804.02  ; RK_05 #2入壳定位陶瓷棒下#2夹紧气缸伸出位标志[0004.02]
AND 804.07  ; RK_05 #2入壳吸盘上#1伸缩气缸缩回位标志[0004.07]
AND 804.08  ; RK_05 #2入壳吸盘上#2伸缩气缸缩回位标志[0004.08]
AND 804.09  ; RK_05 #2入壳吸盘上#3伸缩气缸缩回位标志[0004.09]
AND 804.10  ; RK_05 #2入壳吸盘下#1伸缩气缸缩回位标志[0004.10]
AND 804.11  ; RK_05 #2入壳吸盘下#2伸缩气缸缩回位标志[0004.11]
AND 804.12  ; RK_05 #2入壳吸盘下#3伸缩气缸缩回位标志[0004.12]
AND H36.10  ; RK_05 #2入壳机构立真空记忆
AND 805.13  ; RK_05 #2入壳吸盘真空标志[0005.13]
OUT W227.00  ; RK_05 #2入壳机构入壳条件
; rung 10: #2入壳机构入壳位到待料位条件
LDNOT H36.10  ; RK_05 #2入壳机构立真空记忆
ANDNOT 805.13  ; RK_05 #2入壳吸盘真空标志[0005.13]
AND 804.03  ; RK_05 #2入壳定位陶瓷棒上#1夹紧气缸缩回位标志[0004.03]
AND 804.04  ; RK_05 #2入壳定位陶瓷棒上#2夹紧气缸缩回位标志[0004.04]
AND 804.05  ; RK_05 #2入壳定位陶瓷棒下#1夹紧气缸缩回位标志[0004.05]
AND 804.06  ; RK_05 #2入壳定位陶瓷棒下#2夹紧气缸缩回位标志[0004.06]
AND 801.11  ; RK_05 #2入壳铝壳定位平台升降气缸下降位标志[0001.11]
LD H36.03  ; RK_05 #2入壳机构入壳完成记忆
OR H36.00  ; RK_05 #2入壳机构有电池记忆
ANDLD
ANDNOT H36.04  ; RK_05 #2入壳机构入壳中记忆
ANDNOT H36.01  ; RK_05 #2入壳机构有电芯记忆
LDNOT 805.10  ; RK_05 #2入壳电芯有料感应标志[0005.10]
OR P_On
ANDLD
AND H36.00  ; RK_05 #2入壳机构有电池记忆
ANDNOT H36.02  ; RK_05 #2入壳机构有铝壳记忆
AND 805.11  ; RK_05 #2入壳铝壳有料感应标志[0005.11]
LD H20.00  ; RK_03 U0_U 电芯上料X轴回原点记忆
ANDNOT 853.03  ; RK_03 U0_U 电芯上料X轴#2入壳放料位标志
OR 800.09  ; RK_03 电芯上料升降气缸上升位标志[0000.09]
ANDLD
OUT W227.01  ; RK_05 #2入壳机构入壳位到待料位条件
; rung 11: #2入壳机构工位编号读取
LD D1066.14  ; RK_05 #2入壳机构铝壳定位伸缩气缸伸出1（步）
ANDNOT P_On
OR D1066.13  ; RK_05 #2入壳机构铝壳定位夹爪气缸张开1（步）
OUT TR0
AND P_On
@RSET E2_2800.01  ; #2入壳工位编号标志
LD TR0
@SET E2_2800.01  ; #2入壳工位编号标志

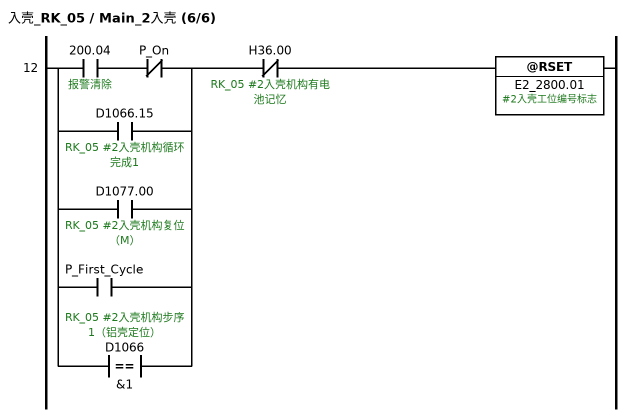
; rung 12
LD 200.04  ; 报警清除
ANDNOT P_On
OR D1066.15  ; RK_05 #2入壳机构循环完成1
OR D1077.00  ; RK_05 #2入壳机构复位（M）
OR P_First_Cycle
OR=(300) D1066 &1  ; RK_05 #2入壳机构步序1（铝壳定位）
ANDNOT H36.00  ; RK_05 #2入壳机构有电池记忆
@RSET E2_2800.01  ; #2入壳工位编号标志

### Section 手动_1入壳

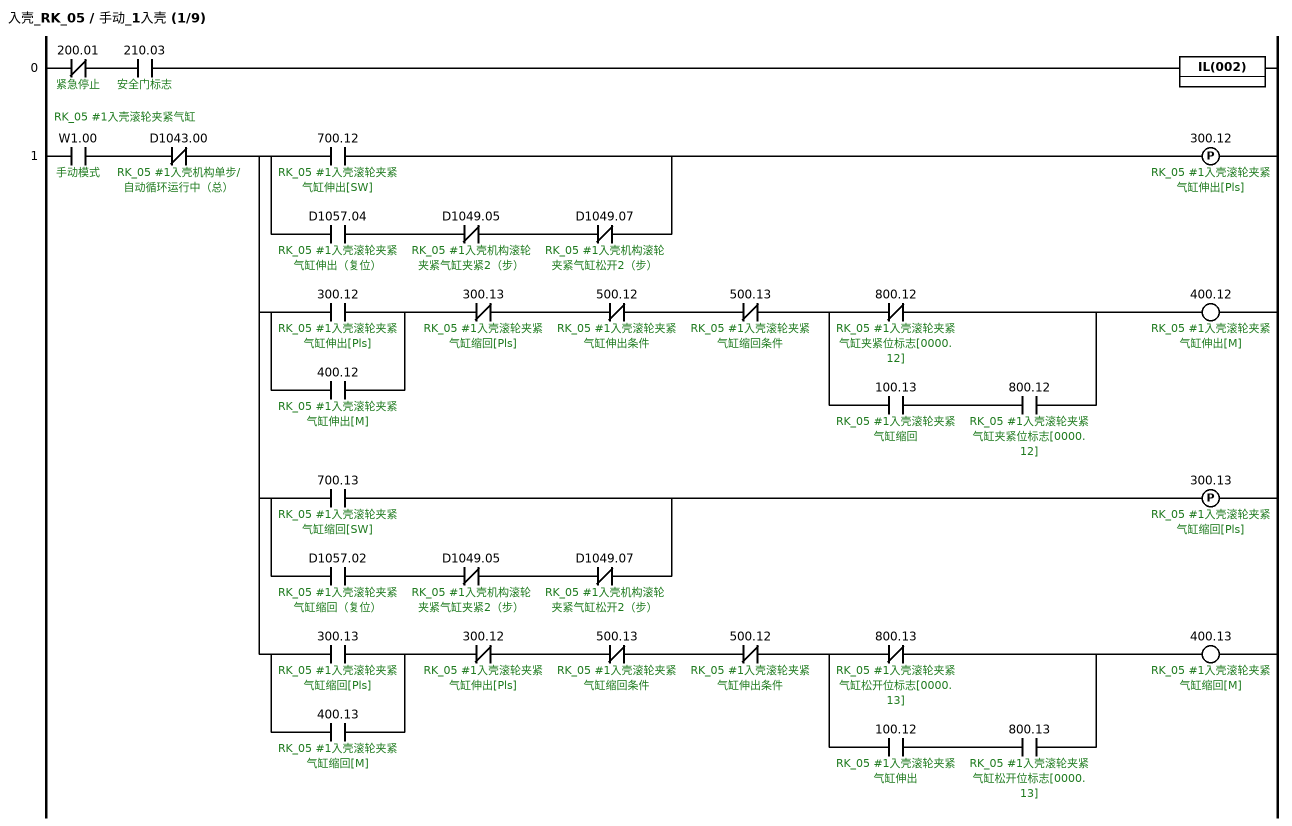
; rung 0
LDNOT 200.01  ; 紧急停止
AND 210.03  ; 安全门标志
IL(002)
; rung 1: RK_05 #1入壳滚轮夹紧气缸
LD W1.00  ; 手动模式
ANDNOT D1043.00  ; RK_05 #1入壳机构单步/自动循环运行中（总）
OUT TR0
LD 700.12  ; RK_05 #1入壳滚轮夹紧气缸伸出[SW]
LD D1057.04  ; RK_05 #1入壳滚轮夹紧气缸伸出（复位）
ANDNOT D1049.05  ; RK_05 #1入壳机构滚轮夹紧气缸夹紧2（步）
ANDNOT D1049.07  ; RK_05 #1入壳机构滚轮夹紧气缸松开2（步）
ORLD
ANDLD
DIFU(013) 300.12  ; RK_05 #1入壳滚轮夹紧气缸伸出[Pls]
LD TR0
LD 300.12  ; RK_05 #1入壳滚轮夹紧气缸伸出[Pls]
OR 400.12  ; RK_05 #1入壳滚轮夹紧气缸伸出[M]
ANDLD
ANDNOT 300.13  ; RK_05 #1入壳滚轮夹紧气缸缩回[Pls]
ANDNOT 500.12  ; RK_05 #1入壳滚轮夹紧气缸伸出条件
ANDNOT 500.13  ; RK_05 #1入壳滚轮夹紧气缸缩回条件
LDNOT 800.12  ; RK_05 #1入壳滚轮夹紧气缸夹紧位标志[0000.12]
LD 100.13  ; RK_05 #1入壳滚轮夹紧气缸缩回
AND 800.12  ; RK_05 #1入壳滚轮夹紧气缸夹紧位标志[0000.12]
ORLD
ANDLD
OUT 400.12  ; RK_05 #1入壳滚轮夹紧气缸伸出[M]
LD TR0
LD 700.13  ; RK_05 #1入壳滚轮夹紧气缸缩回[SW]
LD D1057.02  ; RK_05 #1入壳滚轮夹紧气缸缩回（复位）
ANDNOT D1049.05  ; RK_05 #1入壳机构滚轮夹紧气缸夹紧2（步）
ANDNOT D1049.07  ; RK_05 #1入壳机构滚轮夹紧气缸松开2（步）
ORLD
ANDLD
DIFU(013) 300.13  ; RK_05 #1入壳滚轮夹紧气缸缩回[Pls]
LD TR0
LD 300.13  ; RK_05 #1入壳滚轮夹紧气缸缩回[Pls]
OR 400.13  ; RK_05 #1入壳滚轮夹紧气缸缩回[M]
ANDLD
ANDNOT 300.12  ; RK_05 #1入壳滚轮夹紧气缸伸出[Pls]
ANDNOT 500.13  ; RK_05 #1入壳滚轮夹紧气缸缩回条件
ANDNOT 500.12  ; RK_05 #1入壳滚轮夹紧气缸伸出条件
LDNOT 800.13  ; RK_05 #1入壳滚轮夹紧气缸松开位标志[0000.13]
LD 100.12  ; RK_05 #1入壳滚轮夹紧气缸伸出
AND 800.13  ; RK_05 #1入壳滚轮夹紧气缸松开位标志[0000.13]
ORLD
ANDLD
OUT 400.13  ; RK_05 #1入壳滚轮夹紧气缸缩回[M]

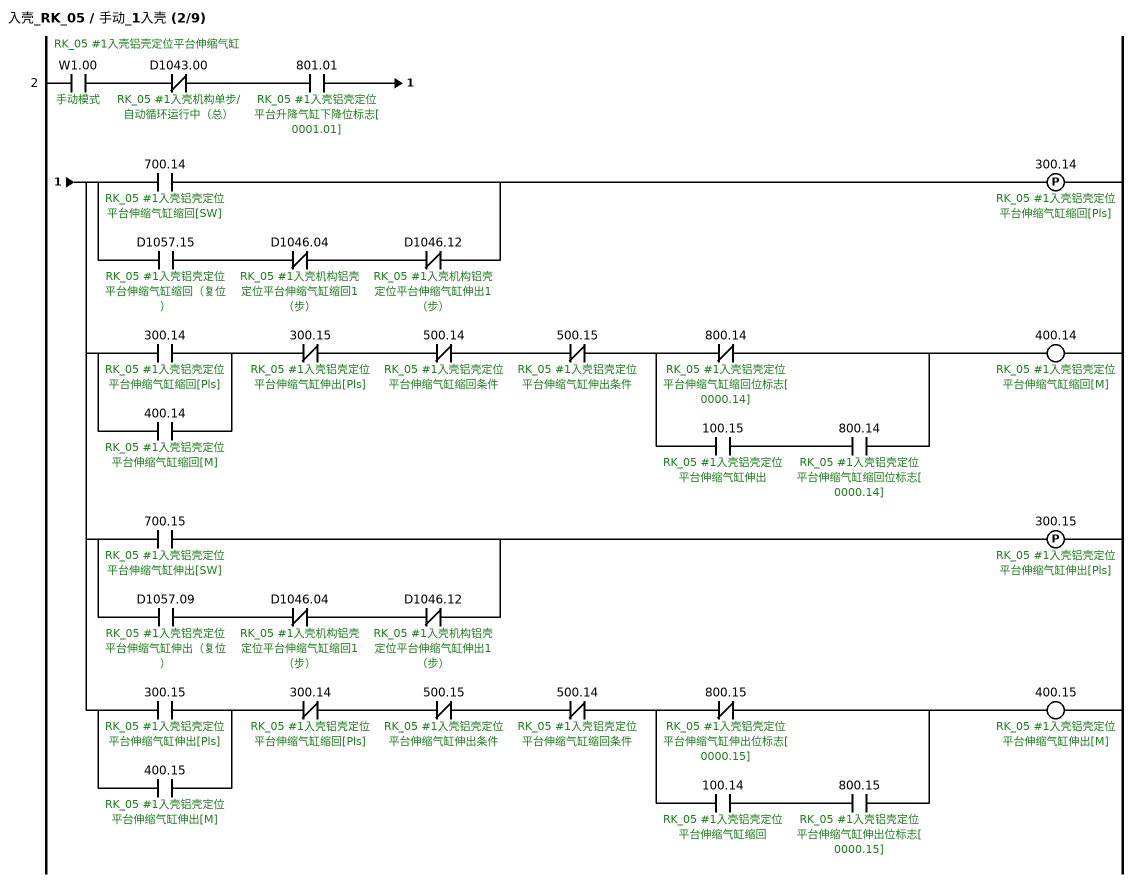
; rung 2: RK_05 #1入壳铝壳定位平台伸缩气缸
LD W1.00  ; 手动模式
ANDNOT D1043.00  ; RK_05 #1入壳机构单步/自动循环运行中（总）
AND 801.01  ; RK_05 #1入壳铝壳定位平台升降气缸下降位标志[0001.01]
OUT TR0
LD 700.14  ; RK_05 #1入壳铝壳定位平台伸缩气缸缩回[SW]
LD D1057.15  ; RK_05 #1入壳铝壳定位平台伸缩气缸缩回（复位）
ANDNOT D1046.04  ; RK_05 #1入壳机构铝壳定位平台伸缩气缸缩回1（步）
ANDNOT D1046.12  ; RK_05 #1入壳机构铝壳定位平台伸缩气缸伸出1（步）
ORLD
ANDLD
DIFU(013) 300.14  ; RK_05 #1入壳铝壳定位平台伸缩气缸缩回[Pls]
LD TR0
LD 300.14  ; RK_05 #1入壳铝壳定位平台伸缩气缸缩回[Pls]
OR 400.14  ; RK_05 #1入壳铝壳定位平台伸缩气缸缩回[M]
ANDLD
ANDNOT 300.15  ; RK_05 #1入壳铝壳定位平台伸缩气缸伸出[Pls]
ANDNOT 500.14  ; RK_05 #1入壳铝壳定位平台伸缩气缸缩回条件
ANDNOT 500.15  ; RK_05 #1入壳铝壳定位平台伸缩气缸伸出条件
LDNOT 800.14  ; RK_05 #1入壳铝壳定位平台伸缩气缸缩回位标志[0000.14]
LD 100.15  ; RK_05 #1入壳铝壳定位平台伸缩气缸伸出
AND 800.14  ; RK_05 #1入壳铝壳定位平台伸缩气缸缩回位标志[0000.14]
ORLD
ANDLD
OUT 400.14  ; RK_05 #1入壳铝壳定位平台伸缩气缸缩回[M]
LD TR0
LD 700.15  ; RK_05 #1入壳铝壳定位平台伸缩气缸伸出[SW]
LD D1057.09  ; RK_05 #1入壳铝壳定位平台伸缩气缸伸出（复位）
ANDNOT D1046.04  ; RK_05 #1入壳机构铝壳定位平台伸缩气缸缩回1（步）
ANDNOT D1046.12  ; RK_05 #1入壳机构铝壳定位平台伸缩气缸伸出1（步）
ORLD
ANDLD
DIFU(013) 300.15  ; RK_05 #1入壳铝壳定位平台伸缩气缸伸出[Pls]
LD TR0
LD 300.15  ; RK_05 #1入壳铝壳定位平台伸缩气缸伸出[Pls]
OR 400.15  ; RK_05 #1入壳铝壳定位平台伸缩气缸伸出[M]
ANDLD
ANDNOT 300.14  ; RK_05 #1入壳铝壳定位平台伸缩气缸缩回[Pls]
ANDNOT 500.15  ; RK_05 #1入壳铝壳定位平台伸缩气缸伸出条件
ANDNOT 500.14  ; RK_05 #1入壳铝壳定位平台伸缩气缸缩回条件
LDNOT 800.15  ; RK_05 #1入壳铝壳定位平台伸缩气缸伸出位标志[0000.15]
LD 100.14  ; RK_05 #1入壳铝壳定位平台伸缩气缸缩回
AND 800.15  ; RK_05 #1入壳铝壳定位平台伸缩气缸伸出位标志[0000.15]
ORLD
ANDLD
OUT 400.15  ; RK_05 #1入壳铝壳定位平台伸缩气缸伸出[M]

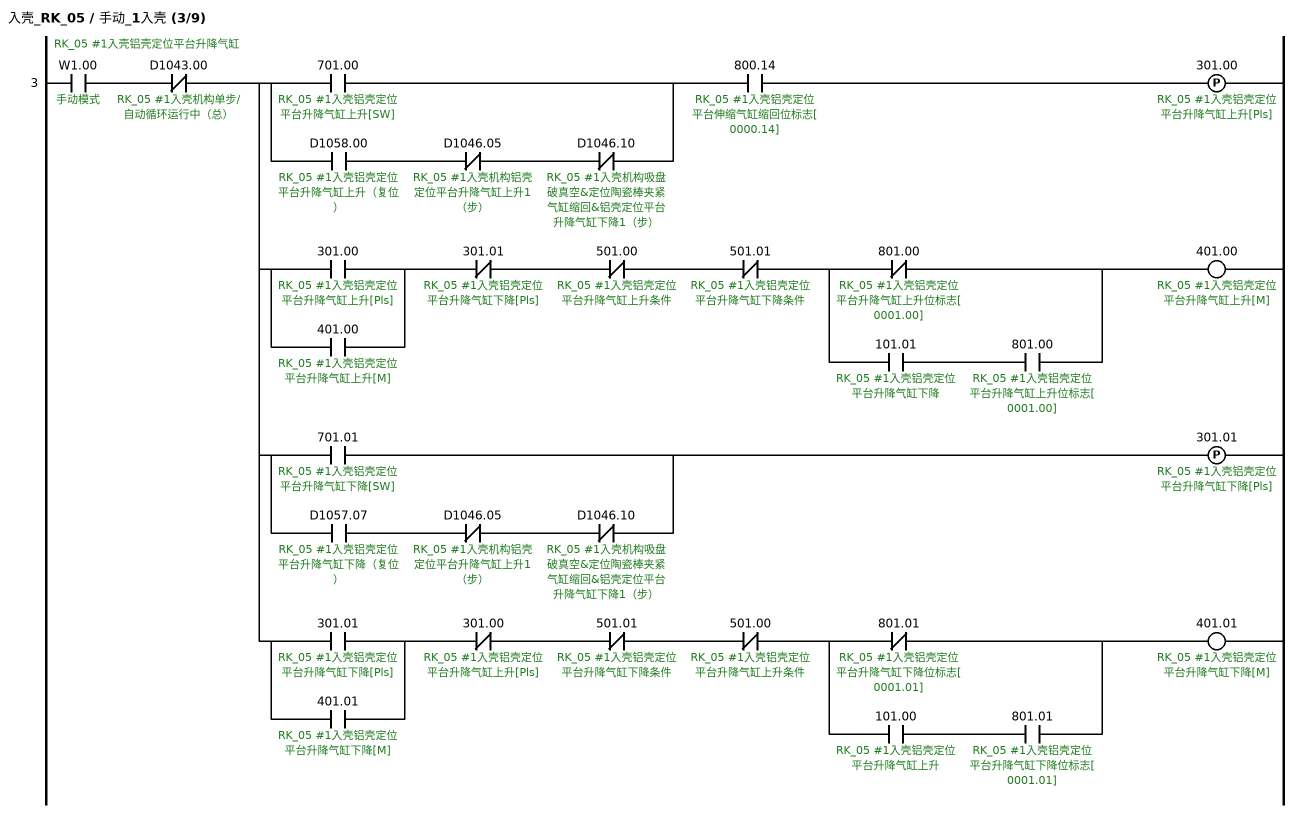
; rung 3: RK_05 #1入壳铝壳定位平台升降气缸
LD W1.00  ; 手动模式
ANDNOT D1043.00  ; RK_05 #1入壳机构单步/自动循环运行中（总）
OUT TR0
LD 701.00  ; RK_05 #1入壳铝壳定位平台升降气缸上升[SW]
LD D1058.00  ; RK_05 #1入壳铝壳定位平台升降气缸上升（复位）
ANDNOT D1046.05  ; RK_05 #1入壳机构铝壳定位平台升降气缸上升1（步）
ANDNOT D1046.10  ; RK_05 #1入壳机构吸盘破真空&定位陶瓷棒夹紧气缸缩回&铝壳定位平台升降气缸下降1（步）
ORLD
ANDLD
AND 800.14  ; RK_05 #1入壳铝壳定位平台伸缩气缸缩回位标志[0000.14]
DIFU(013) 301.00  ; RK_05 #1入壳铝壳定位平台升降气缸上升[Pls]
LD TR0
LD 301.00  ; RK_05 #1入壳铝壳定位平台升降气缸上升[Pls]
OR 401.00  ; RK_05 #1入壳铝壳定位平台升降气缸上升[M]
ANDLD
ANDNOT 301.01  ; RK_05 #1入壳铝壳定位平台升降气缸下降[Pls]
ANDNOT 501.00  ; RK_05 #1入壳铝壳定位平台升降气缸上升条件
ANDNOT 501.01  ; RK_05 #1入壳铝壳定位平台升降气缸下降条件
LDNOT 801.00  ; RK_05 #1入壳铝壳定位平台升降气缸上升位标志[0001.00]
LD 101.01  ; RK_05 #1入壳铝壳定位平台升降气缸下降
AND 801.00  ; RK_05 #1入壳铝壳定位平台升降气缸上升位标志[0001.00]
ORLD
ANDLD
OUT 401.00  ; RK_05 #1入壳铝壳定位平台升降气缸上升[M]
LD TR0
LD 701.01  ; RK_05 #1入壳铝壳定位平台升降气缸下降[SW]
LD D1057.07  ; RK_05 #1入壳铝壳定位平台升降气缸下降（复位）
ANDNOT D1046.05  ; RK_05 #1入壳机构铝壳定位平台升降气缸上升1（步）
ANDNOT D1046.10  ; RK_05 #1入壳机构吸盘破真空&定位陶瓷棒夹紧气缸缩回&铝壳定位平台升降气缸下降1（步）
ORLD
ANDLD
DIFU(013) 301.01  ; RK_05 #1入壳铝壳定位平台升降气缸下降[Pls]
LD TR0
LD 301.01  ; RK_05 #1入壳铝壳定位平台升降气缸下降[Pls]
OR 401.01  ; RK_05 #1入壳铝壳定位平台升降气缸下降[M]
ANDLD
ANDNOT 301.00  ; RK_05 #1入壳铝壳定位平台升降气缸上升[Pls]
ANDNOT 501.01  ; RK_05 #1入壳铝壳定位平台升降气缸下降条件
ANDNOT 501.00  ; RK_05 #1入壳铝壳定位平台升降气缸上升条件
LDNOT 801.01  ; RK_05 #1入壳铝壳定位平台升降气缸下降位标志[0001.01]
LD 101.00  ; RK_05 #1入壳铝壳定位平台升降气缸上升
AND 801.01  ; RK_05 #1入壳铝壳定位平台升降气缸下降位标志[0001.01]
ORLD
ANDLD
OUT 401.01  ; RK_05 #1入壳铝壳定位平台升降气缸下降[M]

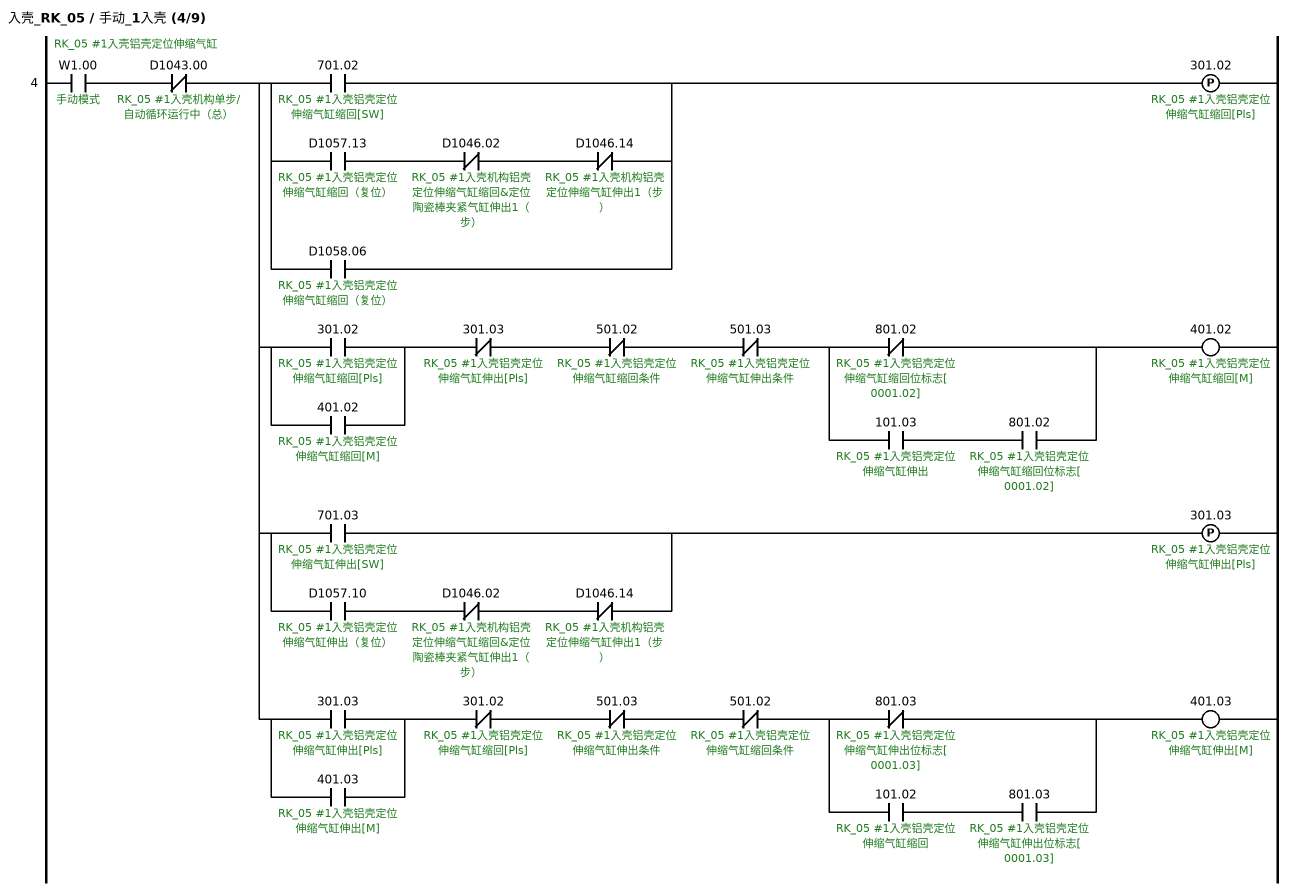
; rung 4: RK_05 #1入壳铝壳定位伸缩气缸
LD W1.00  ; 手动模式
ANDNOT D1043.00  ; RK_05 #1入壳机构单步/自动循环运行中（总）
OUT TR0
LD 701.02  ; RK_05 #1入壳铝壳定位伸缩气缸缩回[SW]
LD D1057.13  ; RK_05 #1入壳铝壳定位伸缩气缸缩回（复位）
ANDNOT D1046.02  ; RK_05 #1入壳机构铝壳定位伸缩气缸缩回&定位陶瓷棒夹紧气缸伸出1（步）
ANDNOT D1046.14  ; RK_05 #1入壳机构铝壳定位伸缩气缸伸出1（步）
ORLD
OR D1058.06  ; RK_05 #1入壳铝壳定位伸缩气缸缩回（复位）
ANDLD
DIFU(013) 301.02  ; RK_05 #1入壳铝壳定位伸缩气缸缩回[Pls]
LD TR0
LD 301.02  ; RK_05 #1入壳铝壳定位伸缩气缸缩回[Pls]
OR 401.02  ; RK_05 #1入壳铝壳定位伸缩气缸缩回[M]
ANDLD
ANDNOT 301.03  ; RK_05 #1入壳铝壳定位伸缩气缸伸出[Pls]
ANDNOT 501.02  ; RK_05 #1入壳铝壳定位伸缩气缸缩回条件
ANDNOT 501.03  ; RK_05 #1入壳铝壳定位伸缩气缸伸出条件
LDNOT 801.02  ; RK_05 #1入壳铝壳定位伸缩气缸缩回位标志[0001.02]
LD 101.03  ; RK_05 #1入壳铝壳定位伸缩气缸伸出
AND 801.02  ; RK_05 #1入壳铝壳定位伸缩气缸缩回位标志[0001.02]
ORLD
ANDLD
OUT 401.02  ; RK_05 #1入壳铝壳定位伸缩气缸缩回[M]
LD TR0
LD 701.03  ; RK_05 #1入壳铝壳定位伸缩气缸伸出[SW]
LD D1057.10  ; RK_05 #1入壳铝壳定位伸缩气缸伸出（复位）
ANDNOT D1046.02  ; RK_05 #1入壳机构铝壳定位伸缩气缸缩回&定位陶瓷棒夹紧气缸伸出1（步）
ANDNOT D1046.14  ; RK_05 #1入壳机构铝壳定位伸缩气缸伸出1（步）
ORLD
ANDLD
DIFU(013) 301.03  ; RK_05 #1入壳铝壳定位伸缩气缸伸出[Pls]
LD TR0
LD 301.03  ; RK_05 #1入壳铝壳定位伸缩气缸伸出[Pls]
OR 401.03  ; RK_05 #1入壳铝壳定位伸缩气缸伸出[M]
ANDLD
ANDNOT 301.02  ; RK_05 #1入壳铝壳定位伸缩气缸缩回[Pls]
ANDNOT 501.03  ; RK_05 #1入壳铝壳定位伸缩气缸伸出条件
ANDNOT 501.02  ; RK_05 #1入壳铝壳定位伸缩气缸缩回条件
LDNOT 801.03  ; RK_05 #1入壳铝壳定位伸缩气缸伸出位标志[0001.03]
LD 101.02  ; RK_05 #1入壳铝壳定位伸缩气缸缩回
AND 801.03  ; RK_05 #1入壳铝壳定位伸缩气缸伸出位标志[0001.03]
ORLD
ANDLD
OUT 401.03  ; RK_05 #1入壳铝壳定位伸缩气缸伸出[M]

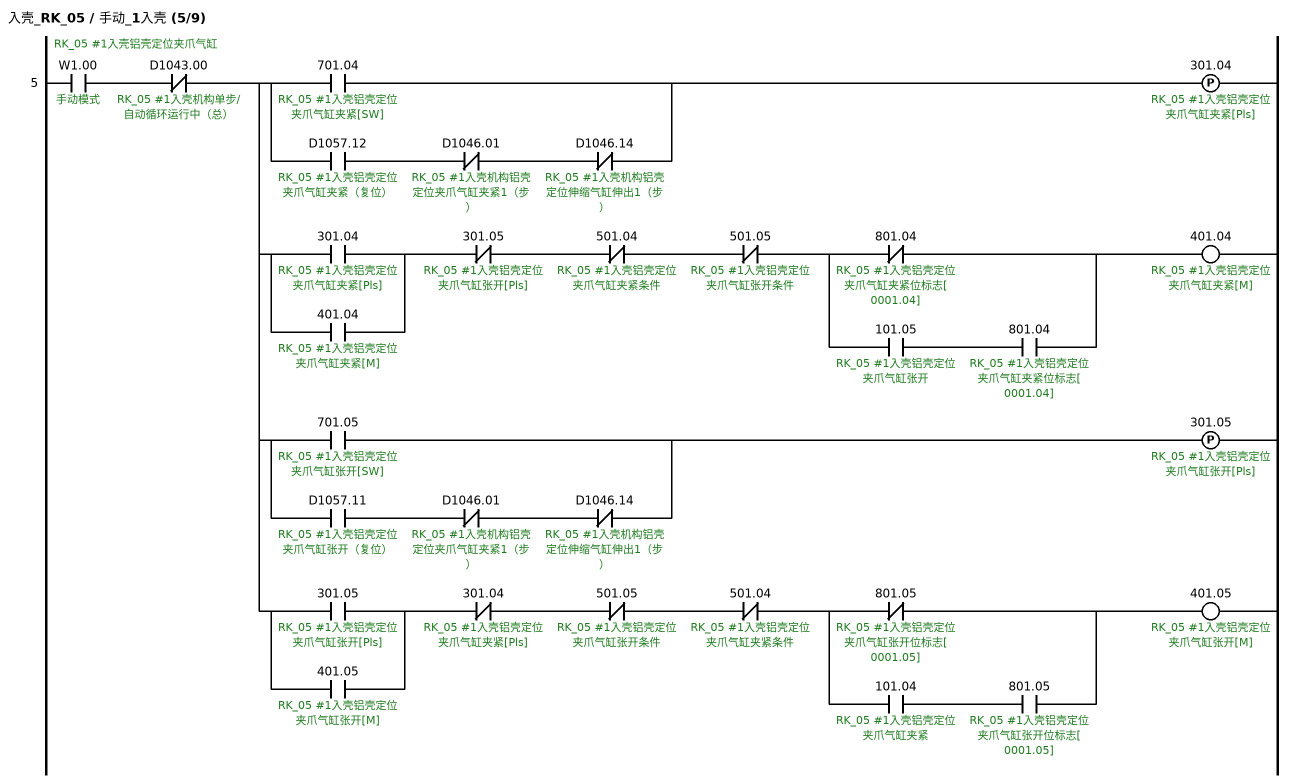
; rung 5: RK_05 #1入壳铝壳定位夹爪气缸
LD W1.00  ; 手动模式
ANDNOT D1043.00  ; RK_05 #1入壳机构单步/自动循环运行中（总）
OUT TR0
LD 701.04  ; RK_05 #1入壳铝壳定位夹爪气缸夹紧[SW]
LD D1057.12  ; RK_05 #1入壳铝壳定位夹爪气缸夹紧（复位）
ANDNOT D1046.01  ; RK_05 #1入壳机构铝壳定位夹爪气缸夹紧1（步）
ANDNOT D1046.14  ; RK_05 #1入壳机构铝壳定位伸缩气缸伸出1（步）
ORLD
ANDLD
DIFU(013) 301.04  ; RK_05 #1入壳铝壳定位夹爪气缸夹紧[Pls]
LD TR0
LD 301.04  ; RK_05 #1入壳铝壳定位夹爪气缸夹紧[Pls]
OR 401.04  ; RK_05 #1入壳铝壳定位夹爪气缸夹紧[M]
ANDLD
ANDNOT 301.05  ; RK_05 #1入壳铝壳定位夹爪气缸张开[Pls]
ANDNOT 501.04  ; RK_05 #1入壳铝壳定位夹爪气缸夹紧条件
ANDNOT 501.05  ; RK_05 #1入壳铝壳定位夹爪气缸张开条件
LDNOT 801.04  ; RK_05 #1入壳铝壳定位夹爪气缸夹紧位标志[0001.04]
LD 101.05  ; RK_05 #1入壳铝壳定位夹爪气缸张开
AND 801.04  ; RK_05 #1入壳铝壳定位夹爪气缸夹紧位标志[0001.04]
ORLD
ANDLD
OUT 401.04  ; RK_05 #1入壳铝壳定位夹爪气缸夹紧[M]
LD TR0
LD 701.05  ; RK_05 #1入壳铝壳定位夹爪气缸张开[SW]
LD D1057.11  ; RK_05 #1入壳铝壳定位夹爪气缸张开（复位）
ANDNOT D1046.01  ; RK_05 #1入壳机构铝壳定位夹爪气缸夹紧1（步）
ANDNOT D1046.14  ; RK_05 #1入壳机构铝壳定位伸缩气缸伸出1（步）
ORLD
ANDLD
DIFU(013) 301.05  ; RK_05 #1入壳铝壳定位夹爪气缸张开[Pls]
LD TR0
LD 301.05  ; RK_05 #1入壳铝壳定位夹爪气缸张开[Pls]
OR 401.05  ; RK_05 #1入壳铝壳定位夹爪气缸张开[M]
ANDLD
ANDNOT 301.04  ; RK_05 #1入壳铝壳定位夹爪气缸夹紧[Pls]
ANDNOT 501.05  ; RK_05 #1入壳铝壳定位夹爪气缸张开条件
ANDNOT 501.04  ; RK_05 #1入壳铝壳定位夹爪气缸夹紧条件
LDNOT 801.05  ; RK_05 #1入壳铝壳定位夹爪气缸张开位标志[0001.05]
LD 101.04  ; RK_05 #1入壳铝壳定位夹爪气缸夹紧
AND 801.05  ; RK_05 #1入壳铝壳定位夹爪气缸张开位标志[0001.05]
ORLD
ANDLD
OUT 401.05  ; RK_05 #1入壳铝壳定位夹爪气缸张开[M]

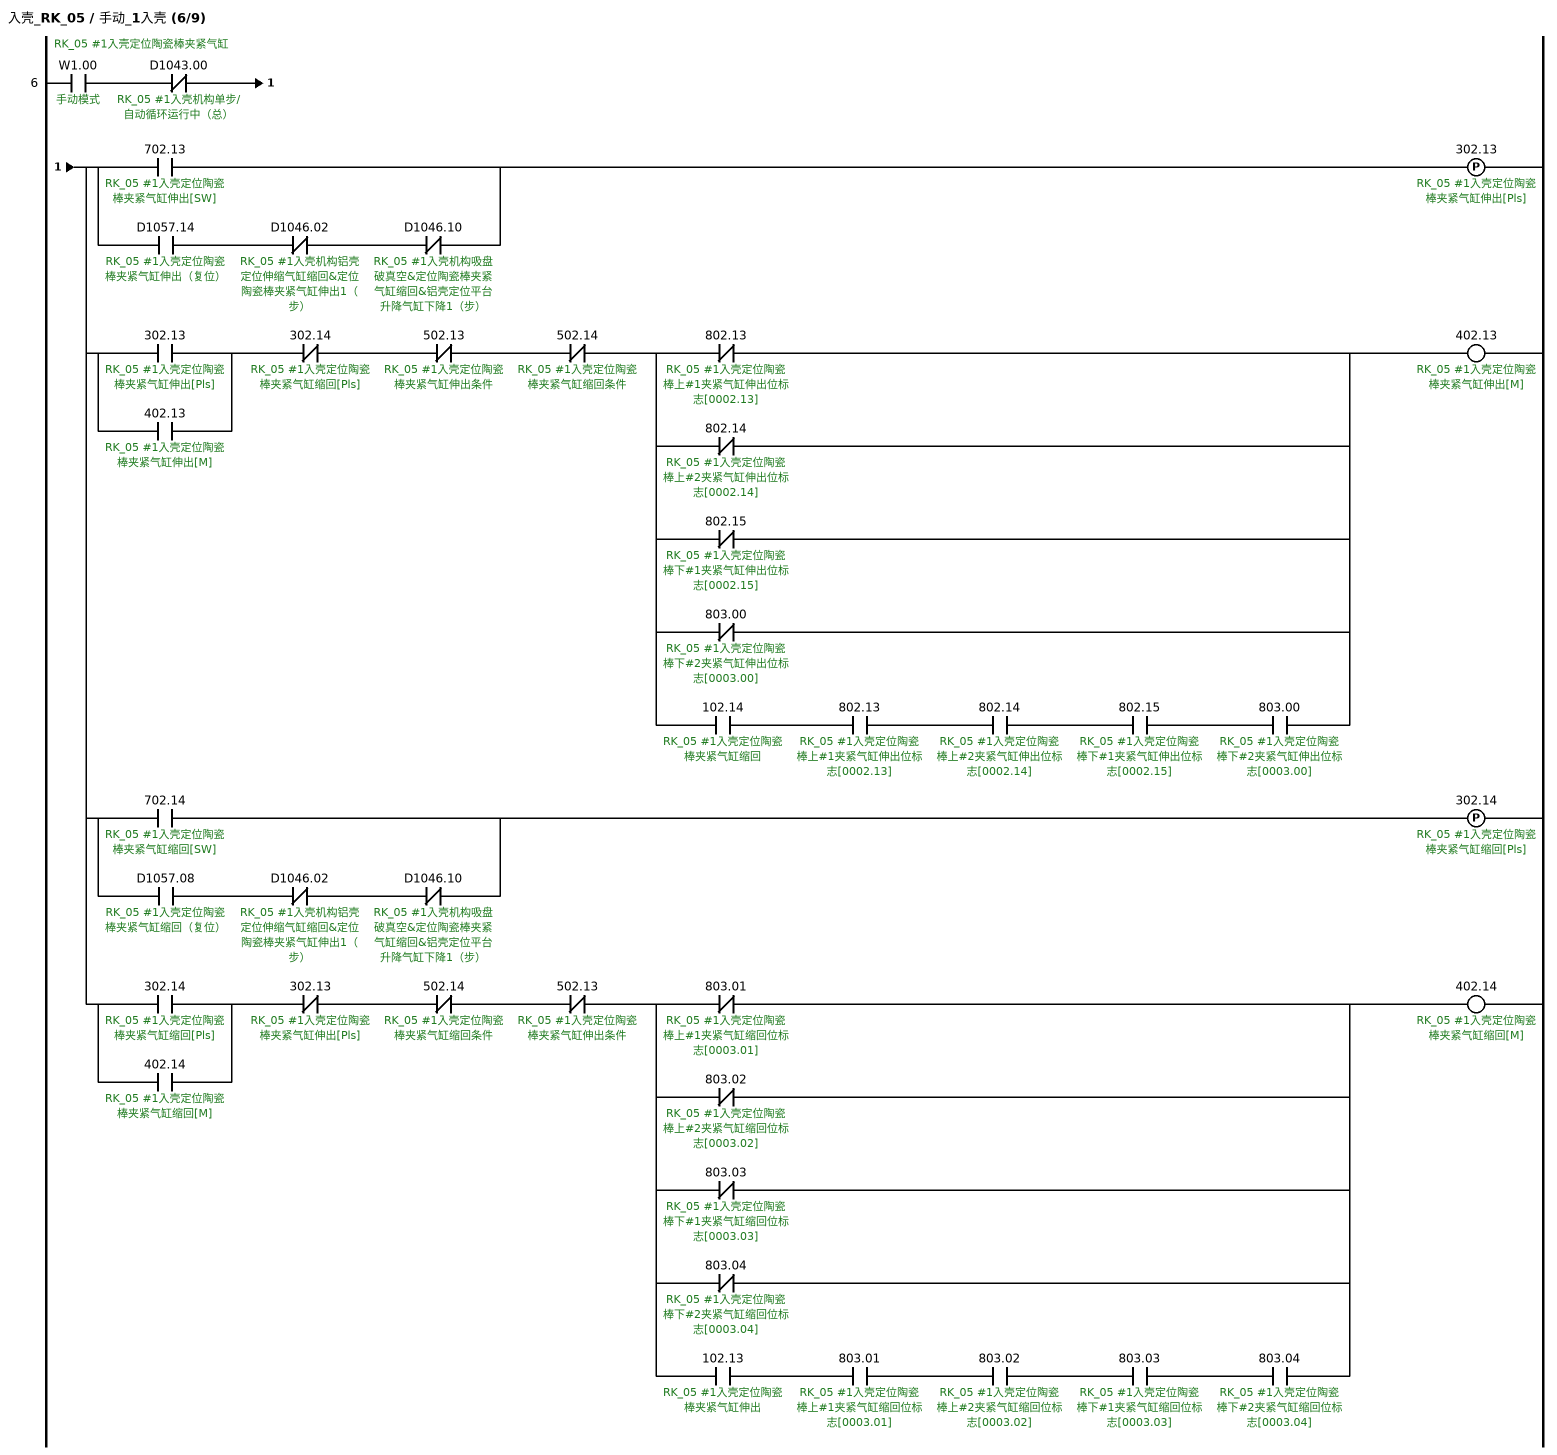
; rung 6: RK_05 #1入壳定位陶瓷棒夹紧气缸
LD W1.00  ; 手动模式
ANDNOT D1043.00  ; RK_05 #1入壳机构单步/自动循环运行中（总）
OUT TR0
LD 702.13  ; RK_05 #1入壳定位陶瓷棒夹紧气缸伸出[SW]
LD D1057.14  ; RK_05 #1入壳定位陶瓷棒夹紧气缸伸出（复位）
ANDNOT D1046.02  ; RK_05 #1入壳机构铝壳定位伸缩气缸缩回&定位陶瓷棒夹紧气缸伸出1（步）
ANDNOT D1046.10  ; RK_05 #1入壳机构吸盘破真空&定位陶瓷棒夹紧气缸缩回&铝壳定位平台升降气缸下降1（步）
ORLD
ANDLD
DIFU(013) 302.13  ; RK_05 #1入壳定位陶瓷棒夹紧气缸伸出[Pls]
LD TR0
LD 302.13  ; RK_05 #1入壳定位陶瓷棒夹紧气缸伸出[Pls]
OR 402.13  ; RK_05 #1入壳定位陶瓷棒夹紧气缸伸出[M]
ANDLD
ANDNOT 302.14  ; RK_05 #1入壳定位陶瓷棒夹紧气缸缩回[Pls]
ANDNOT 502.13  ; RK_05 #1入壳定位陶瓷棒夹紧气缸伸出条件
ANDNOT 502.14  ; RK_05 #1入壳定位陶瓷棒夹紧气缸缩回条件
LDNOT 802.13  ; RK_05 #1入壳定位陶瓷棒上#1夹紧气缸伸出位标志[0002.13]
ORNOT 802.14  ; RK_05 #1入壳定位陶瓷棒上#2夹紧气缸伸出位标志[0002.14]
ORNOT 802.15  ; RK_05 #1入壳定位陶瓷棒下#1夹紧气缸伸出位标志[0002.15]
ORNOT 803.00  ; RK_05 #1入壳定位陶瓷棒下#2夹紧气缸伸出位标志[0003.00]
LD 102.14  ; RK_05 #1入壳定位陶瓷棒夹紧气缸缩回
AND 802.13  ; RK_05 #1入壳定位陶瓷棒上#1夹紧气缸伸出位标志[0002.13]
AND 802.14  ; RK_05 #1入壳定位陶瓷棒上#2夹紧气缸伸出位标志[0002.14]
AND 802.15  ; RK_05 #1入壳定位陶瓷棒下#1夹紧气缸伸出位标志[0002.15]
AND 803.00  ; RK_05 #1入壳定位陶瓷棒下#2夹紧气缸伸出位标志[0003.00]
ORLD
ANDLD
OUT 402.13  ; RK_05 #1入壳定位陶瓷棒夹紧气缸伸出[M]
LD TR0
LD 702.14  ; RK_05 #1入壳定位陶瓷棒夹紧气缸缩回[SW]
LD D1057.08  ; RK_05 #1入壳定位陶瓷棒夹紧气缸缩回（复位）
ANDNOT D1046.02  ; RK_05 #1入壳机构铝壳定位伸缩气缸缩回&定位陶瓷棒夹紧气缸伸出1（步）
ANDNOT D1046.10  ; RK_05 #1入壳机构吸盘破真空&定位陶瓷棒夹紧气缸缩回&铝壳定位平台升降气缸下降1（步）
ORLD
ANDLD
DIFU(013) 302.14  ; RK_05 #1入壳定位陶瓷棒夹紧气缸缩回[Pls]
LD TR0
LD 302.14  ; RK_05 #1入壳定位陶瓷棒夹紧气缸缩回[Pls]
OR 402.14  ; RK_05 #1入壳定位陶瓷棒夹紧气缸缩回[M]
ANDLD
ANDNOT 302.13  ; RK_05 #1入壳定位陶瓷棒夹紧气缸伸出[Pls]
ANDNOT 502.14  ; RK_05 #1入壳定位陶瓷棒夹紧气缸缩回条件
ANDNOT 502.13  ; RK_05 #1入壳定位陶瓷棒夹紧气缸伸出条件
LDNOT 803.01  ; RK_05 #1入壳定位陶瓷棒上#1夹紧气缸缩回位标志[0003.01]
ORNOT 803.02  ; RK_05 #1入壳定位陶瓷棒上#2夹紧气缸缩回位标志[0003.02]
ORNOT 803.03  ; RK_05 #1入壳定位陶瓷棒下#1夹紧气缸缩回位标志[0003.03]
ORNOT 803.04  ; RK_05 #1入壳定位陶瓷棒下#2夹紧气缸缩回位标志[0003.04]
LD 102.13  ; RK_05 #1入壳定位陶瓷棒夹紧气缸伸出
AND 803.01  ; RK_05 #1入壳定位陶瓷棒上#1夹紧气缸缩回位标志[0003.01]
AND 803.02  ; RK_05 #1入壳定位陶瓷棒上#2夹紧气缸缩回位标志[0003.02]
AND 803.03  ; RK_05 #1入壳定位陶瓷棒下#1夹紧气缸缩回位标志[0003.03]
AND 803.04  ; RK_05 #1入壳定位陶瓷棒下#2夹紧气缸缩回位标志[0003.04]
ORLD
ANDLD
OUT 402.14  ; RK_05 #1入壳定位陶瓷棒夹紧气缸缩回[M]

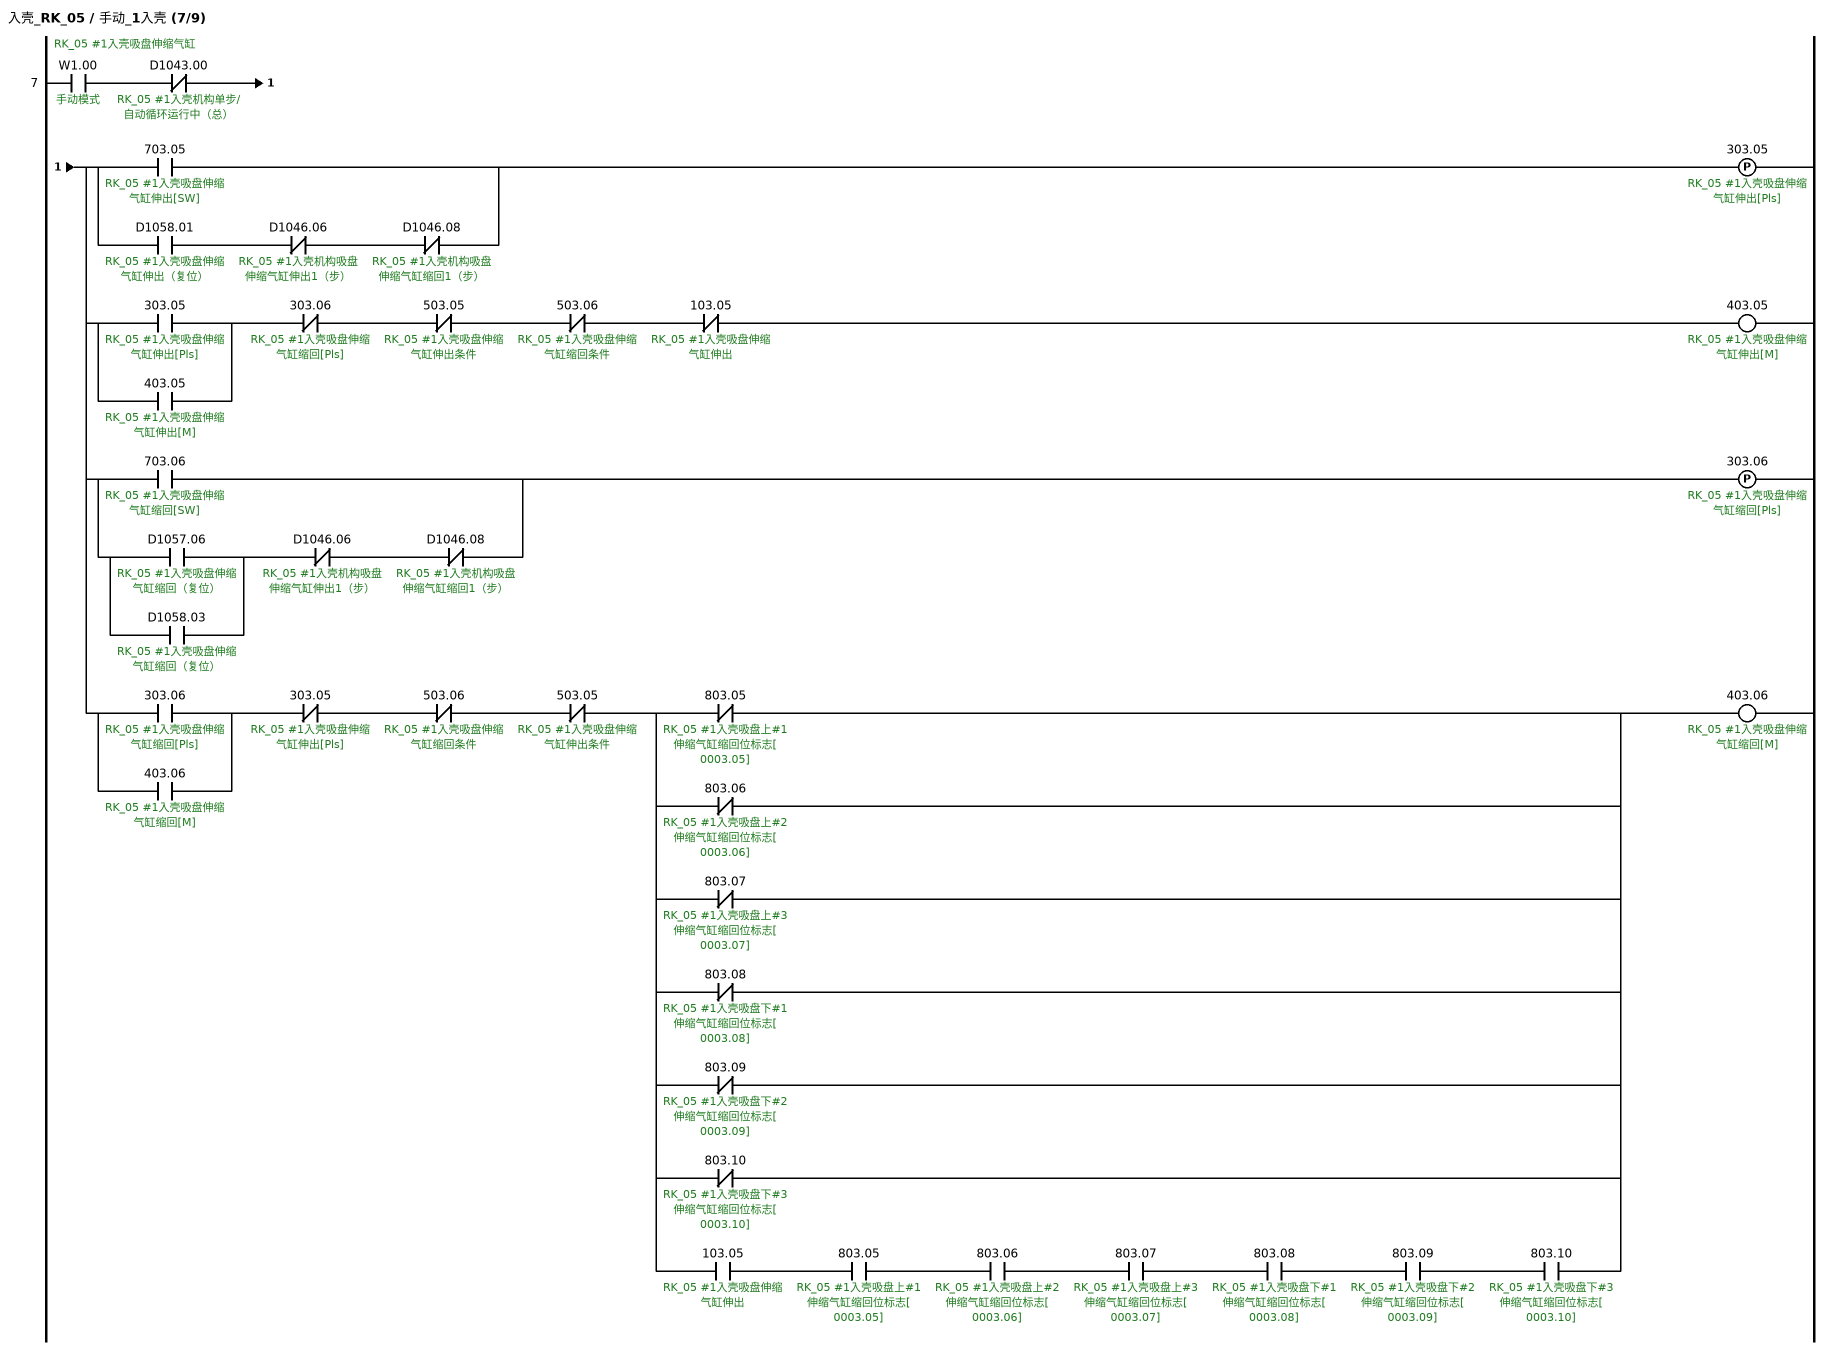
; rung 7: RK_05 #1入壳吸盘伸缩气缸
LD W1.00  ; 手动模式
ANDNOT D1043.00  ; RK_05 #1入壳机构单步/自动循环运行中（总）
OUT TR0
LD 703.05  ; RK_05 #1入壳吸盘伸缩气缸伸出[SW]
LD D1058.01  ; RK_05 #1入壳吸盘伸缩气缸伸出（复位）
ANDNOT D1046.06  ; RK_05 #1入壳机构吸盘伸缩气缸伸出1（步）
ANDNOT D1046.08  ; RK_05 #1入壳机构吸盘伸缩气缸缩回1（步）
ORLD
ANDLD
DIFU(013) 303.05  ; RK_05 #1入壳吸盘伸缩气缸伸出[Pls]
LD TR0
LD 303.05  ; RK_05 #1入壳吸盘伸缩气缸伸出[Pls]
OR 403.05  ; RK_05 #1入壳吸盘伸缩气缸伸出[M]
ANDLD
ANDNOT 303.06  ; RK_05 #1入壳吸盘伸缩气缸缩回[Pls]
ANDNOT 503.05  ; RK_05 #1入壳吸盘伸缩气缸伸出条件
ANDNOT 503.06  ; RK_05 #1入壳吸盘伸缩气缸缩回条件
ANDNOT 103.05  ; RK_05 #1入壳吸盘伸缩气缸伸出
OUT 403.05  ; RK_05 #1入壳吸盘伸缩气缸伸出[M]
LD TR0
LD 703.06  ; RK_05 #1入壳吸盘伸缩气缸缩回[SW]
LD D1057.06  ; RK_05 #1入壳吸盘伸缩气缸缩回（复位）
OR D1058.03  ; RK_05 #1入壳吸盘伸缩气缸缩回（复位）
ANDNOT D1046.06  ; RK_05 #1入壳机构吸盘伸缩气缸伸出1（步）
ANDNOT D1046.08  ; RK_05 #1入壳机构吸盘伸缩气缸缩回1（步）
ORLD
ANDLD
DIFU(013) 303.06  ; RK_05 #1入壳吸盘伸缩气缸缩回[Pls]
LD TR0
LD 303.06  ; RK_05 #1入壳吸盘伸缩气缸缩回[Pls]
OR 403.06  ; RK_05 #1入壳吸盘伸缩气缸缩回[M]
ANDLD
ANDNOT 303.05  ; RK_05 #1入壳吸盘伸缩气缸伸出[Pls]
ANDNOT 503.06  ; RK_05 #1入壳吸盘伸缩气缸缩回条件
ANDNOT 503.05  ; RK_05 #1入壳吸盘伸缩气缸伸出条件
LDNOT 803.05  ; RK_05 #1入壳吸盘上#1伸缩气缸缩回位标志[0003.05]
ORNOT 803.06  ; RK_05 #1入壳吸盘上#2伸缩气缸缩回位标志[0003.06]
ORNOT 803.07  ; RK_05 #1入壳吸盘上#3伸缩气缸缩回位标志[0003.07]
ORNOT 803.08  ; RK_05 #1入壳吸盘下#1伸缩气缸缩回位标志[0003.08]
ORNOT 803.09  ; RK_05 #1入壳吸盘下#2伸缩气缸缩回位标志[0003.09]
ORNOT 803.10  ; RK_05 #1入壳吸盘下#3伸缩气缸缩回位标志[0003.10]
LD 103.05  ; RK_05 #1入壳吸盘伸缩气缸伸出
AND 803.05  ; RK_05 #1入壳吸盘上#1伸缩气缸缩回位标志[0003.05]
AND 803.06  ; RK_05 #1入壳吸盘上#2伸缩气缸缩回位标志[0003.06]
AND 803.07  ; RK_05 #1入壳吸盘上#3伸缩气缸缩回位标志[0003.07]
AND 803.08  ; RK_05 #1入壳吸盘下#1伸缩气缸缩回位标志[0003.08]
AND 803.09  ; RK_05 #1入壳吸盘下#2伸缩气缸缩回位标志[0003.09]
AND 803.10  ; RK_05 #1入壳吸盘下#3伸缩气缸缩回位标志[0003.10]
ORLD
ANDLD
OUT 403.06  ; RK_05 #1入壳吸盘伸缩气缸缩回[M]

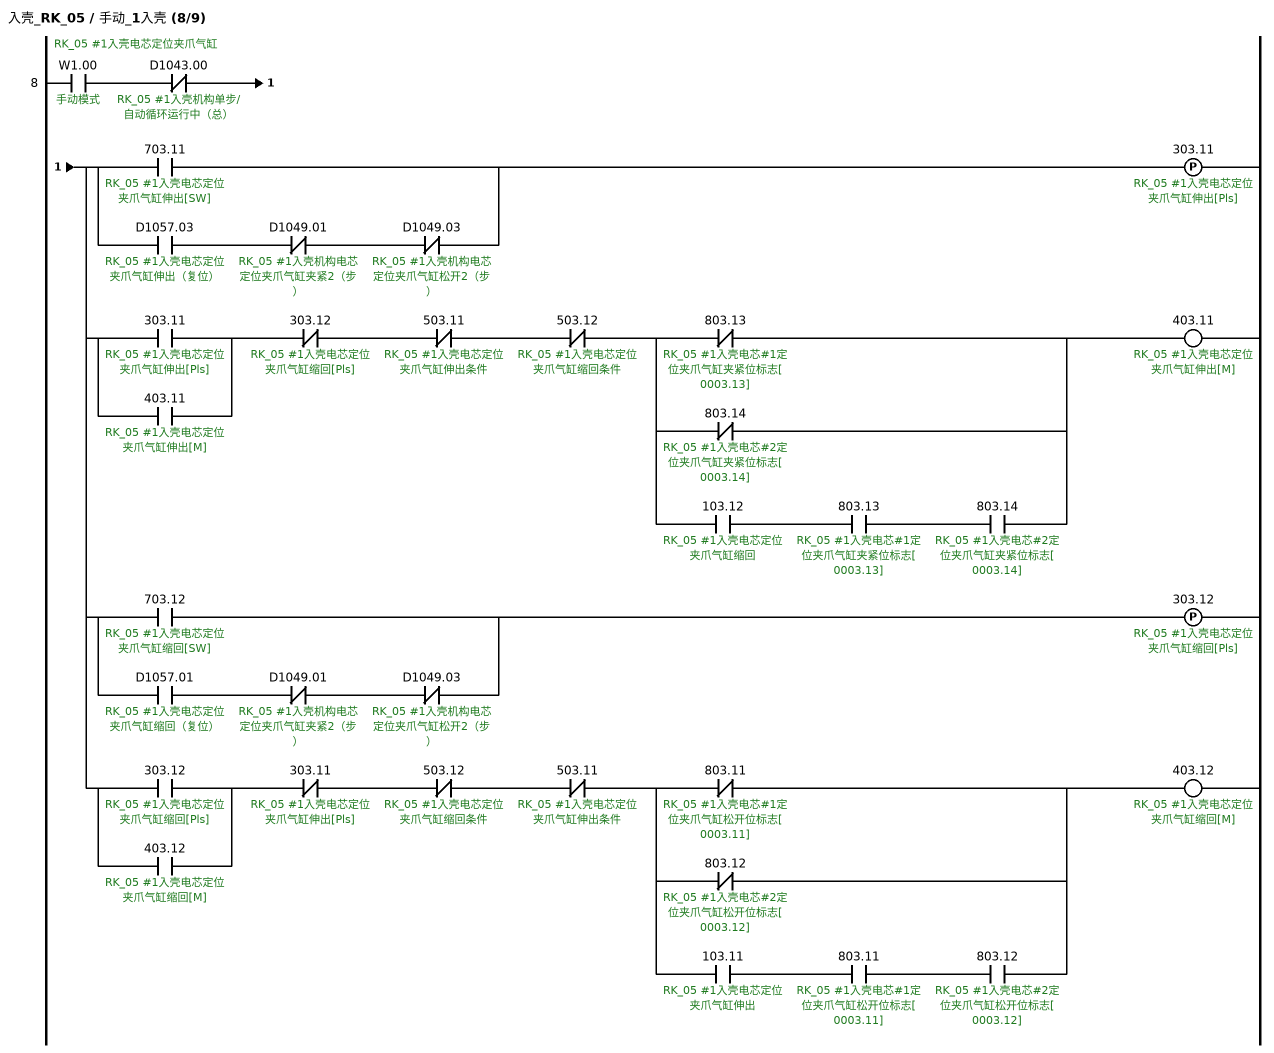
; rung 8: RK_05 #1入壳电芯定位夹爪气缸
LD W1.00  ; 手动模式
ANDNOT D1043.00  ; RK_05 #1入壳机构单步/自动循环运行中（总）
OUT TR0
LD 703.11  ; RK_05 #1入壳电芯定位夹爪气缸伸出[SW]
LD D1057.03  ; RK_05 #1入壳电芯定位夹爪气缸伸出（复位）
ANDNOT D1049.01  ; RK_05 #1入壳机构电芯定位夹爪气缸夹紧2（步）
ANDNOT D1049.03  ; RK_05 #1入壳机构电芯定位夹爪气缸松开2（步）
ORLD
ANDLD
DIFU(013) 303.11  ; RK_05 #1入壳电芯定位夹爪气缸伸出[Pls]
LD TR0
LD 303.11  ; RK_05 #1入壳电芯定位夹爪气缸伸出[Pls]
OR 403.11  ; RK_05 #1入壳电芯定位夹爪气缸伸出[M]
ANDLD
ANDNOT 303.12  ; RK_05 #1入壳电芯定位夹爪气缸缩回[Pls]
ANDNOT 503.11  ; RK_05 #1入壳电芯定位夹爪气缸伸出条件
ANDNOT 503.12  ; RK_05 #1入壳电芯定位夹爪气缸缩回条件
LDNOT 803.13  ; RK_05 #1入壳电芯#1定位夹爪气缸夹紧位标志[0003.13]
ORNOT 803.14  ; RK_05 #1入壳电芯#2定位夹爪气缸夹紧位标志[0003.14]
LD 103.12  ; RK_05 #1入壳电芯定位夹爪气缸缩回
AND 803.13  ; RK_05 #1入壳电芯#1定位夹爪气缸夹紧位标志[0003.13]
AND 803.14  ; RK_05 #1入壳电芯#2定位夹爪气缸夹紧位标志[0003.14]
ORLD
ANDLD
OUT 403.11  ; RK_05 #1入壳电芯定位夹爪气缸伸出[M]
LD TR0
LD 703.12  ; RK_05 #1入壳电芯定位夹爪气缸缩回[SW]
LD D1057.01  ; RK_05 #1入壳电芯定位夹爪气缸缩回（复位）
ANDNOT D1049.01  ; RK_05 #1入壳机构电芯定位夹爪气缸夹紧2（步）
ANDNOT D1049.03  ; RK_05 #1入壳机构电芯定位夹爪气缸松开2（步）
ORLD
ANDLD
DIFU(013) 303.12  ; RK_05 #1入壳电芯定位夹爪气缸缩回[Pls]
LD TR0
LD 303.12  ; RK_05 #1入壳电芯定位夹爪气缸缩回[Pls]
OR 403.12  ; RK_05 #1入壳电芯定位夹爪气缸缩回[M]
ANDLD
ANDNOT 303.11  ; RK_05 #1入壳电芯定位夹爪气缸伸出[Pls]
ANDNOT 503.12  ; RK_05 #1入壳电芯定位夹爪气缸缩回条件
ANDNOT 503.11  ; RK_05 #1入壳电芯定位夹爪气缸伸出条件
LDNOT 803.11  ; RK_05 #1入壳电芯#1定位夹爪气缸松开位标志[0003.11]
ORNOT 803.12  ; RK_05 #1入壳电芯#2定位夹爪气缸松开位标志[0003.12]
LD 103.11  ; RK_05 #1入壳电芯定位夹爪气缸伸出
AND 803.11  ; RK_05 #1入壳电芯#1定位夹爪气缸松开位标志[0003.11]
AND 803.12  ; RK_05 #1入壳电芯#2定位夹爪气缸松开位标志[0003.12]
ORLD
ANDLD
OUT 403.12  ; RK_05 #1入壳电芯定位夹爪气缸缩回[M]

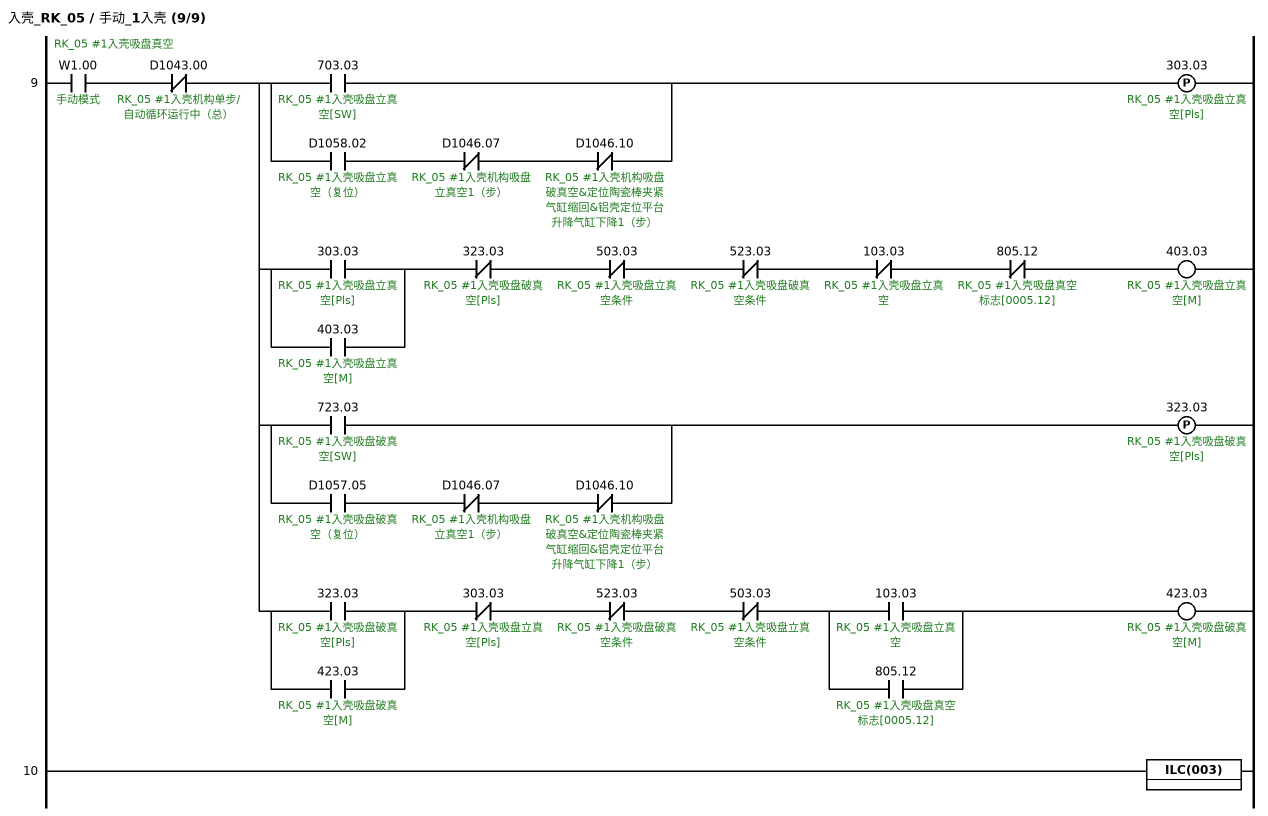
; rung 9: RK_05 #1入壳吸盘真空
LD W1.00  ; 手动模式
ANDNOT D1043.00  ; RK_05 #1入壳机构单步/自动循环运行中（总）
OUT TR0
LD 703.03  ; RK_05 #1入壳吸盘立真空[SW]
LD D1058.02  ; RK_05 #1入壳吸盘立真空（复位）
ANDNOT D1046.07  ; RK_05 #1入壳机构吸盘立真空1（步）
ANDNOT D1046.10  ; RK_05 #1入壳机构吸盘破真空&定位陶瓷棒夹紧气缸缩回&铝壳定位平台升降气缸下降1（步）
ORLD
ANDLD
DIFU(013) 303.03  ; RK_05 #1入壳吸盘立真空[Pls]
LD TR0
LD 303.03  ; RK_05 #1入壳吸盘立真空[Pls]
OR 403.03  ; RK_05 #1入壳吸盘立真空[M]
ANDLD
ANDNOT 323.03  ; RK_05 #1入壳吸盘破真空[Pls]
ANDNOT 503.03  ; RK_05 #1入壳吸盘立真空条件
ANDNOT 523.03  ; RK_05 #1入壳吸盘破真空条件
ANDNOT 103.03  ; RK_05 #1入壳吸盘立真空
ANDNOT 805.12  ; RK_05 #1入壳吸盘真空标志[0005.12]
OUT 403.03  ; RK_05 #1入壳吸盘立真空[M]
LD TR0
LD 723.03  ; RK_05 #1入壳吸盘破真空[SW]
LD D1057.05  ; RK_05 #1入壳吸盘破真空（复位）
ANDNOT D1046.07  ; RK_05 #1入壳机构吸盘立真空1（步）
ANDNOT D1046.10  ; RK_05 #1入壳机构吸盘破真空&定位陶瓷棒夹紧气缸缩回&铝壳定位平台升降气缸下降1（步）
ORLD
ANDLD
DIFU(013) 323.03  ; RK_05 #1入壳吸盘破真空[Pls]
LD TR0
LD 323.03  ; RK_05 #1入壳吸盘破真空[Pls]
OR 423.03  ; RK_05 #1入壳吸盘破真空[M]
ANDLD
ANDNOT 303.03  ; RK_05 #1入壳吸盘立真空[Pls]
ANDNOT 523.03  ; RK_05 #1入壳吸盘破真空条件
ANDNOT 503.03  ; RK_05 #1入壳吸盘立真空条件
LD 103.03  ; RK_05 #1入壳吸盘立真空
OR 805.12  ; RK_05 #1入壳吸盘真空标志[0005.12]
ANDLD
OUT 423.03  ; RK_05 #1入壳吸盘破真空[M]
; rung 10
ILC(003)

### Section 手动_2入壳

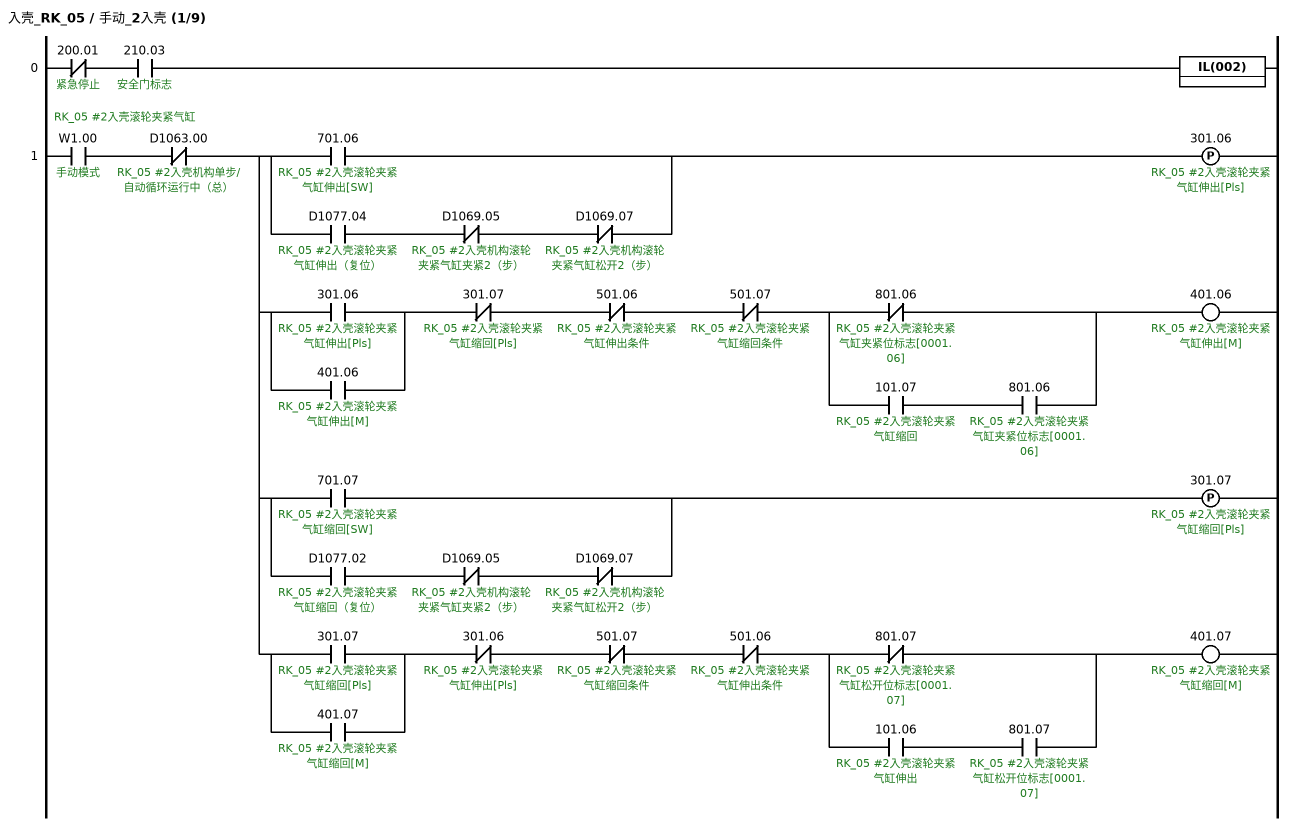
; rung 0
LDNOT 200.01  ; 紧急停止
AND 210.03  ; 安全门标志
IL(002)
; rung 1: RK_05 #2入壳滚轮夹紧气缸
LD W1.00  ; 手动模式
ANDNOT D1063.00  ; RK_05 #2入壳机构单步/自动循环运行中（总）
OUT TR0
LD 701.06  ; RK_05 #2入壳滚轮夹紧气缸伸出[SW]
LD D1077.04  ; RK_05 #2入壳滚轮夹紧气缸伸出（复位）
ANDNOT D1069.05  ; RK_05 #2入壳机构滚轮夹紧气缸夹紧2（步）
ANDNOT D1069.07  ; RK_05 #2入壳机构滚轮夹紧气缸松开2（步）
ORLD
ANDLD
DIFU(013) 301.06  ; RK_05 #2入壳滚轮夹紧气缸伸出[Pls]
LD TR0
LD 301.06  ; RK_05 #2入壳滚轮夹紧气缸伸出[Pls]
OR 401.06  ; RK_05 #2入壳滚轮夹紧气缸伸出[M]
ANDLD
ANDNOT 301.07  ; RK_05 #2入壳滚轮夹紧气缸缩回[Pls]
ANDNOT 501.06  ; RK_05 #2入壳滚轮夹紧气缸伸出条件
ANDNOT 501.07  ; RK_05 #2入壳滚轮夹紧气缸缩回条件
LDNOT 801.06  ; RK_05 #2入壳滚轮夹紧气缸夹紧位标志[0001.06]
LD 101.07  ; RK_05 #2入壳滚轮夹紧气缸缩回
AND 801.06  ; RK_05 #2入壳滚轮夹紧气缸夹紧位标志[0001.06]
ORLD
ANDLD
OUT 401.06  ; RK_05 #2入壳滚轮夹紧气缸伸出[M]
LD TR0
LD 701.07  ; RK_05 #2入壳滚轮夹紧气缸缩回[SW]
LD D1077.02  ; RK_05 #2入壳滚轮夹紧气缸缩回（复位）
ANDNOT D1069.05  ; RK_05 #2入壳机构滚轮夹紧气缸夹紧2（步）
ANDNOT D1069.07  ; RK_05 #2入壳机构滚轮夹紧气缸松开2（步）
ORLD
ANDLD
DIFU(013) 301.07  ; RK_05 #2入壳滚轮夹紧气缸缩回[Pls]
LD TR0
LD 301.07  ; RK_05 #2入壳滚轮夹紧气缸缩回[Pls]
OR 401.07  ; RK_05 #2入壳滚轮夹紧气缸缩回[M]
ANDLD
ANDNOT 301.06  ; RK_05 #2入壳滚轮夹紧气缸伸出[Pls]
ANDNOT 501.07  ; RK_05 #2入壳滚轮夹紧气缸缩回条件
ANDNOT 501.06  ; RK_05 #2入壳滚轮夹紧气缸伸出条件
LDNOT 801.07  ; RK_05 #2入壳滚轮夹紧气缸松开位标志[0001.07]
LD 101.06  ; RK_05 #2入壳滚轮夹紧气缸伸出
AND 801.07  ; RK_05 #2入壳滚轮夹紧气缸松开位标志[0001.07]
ORLD
ANDLD
OUT 401.07  ; RK_05 #2入壳滚轮夹紧气缸缩回[M]

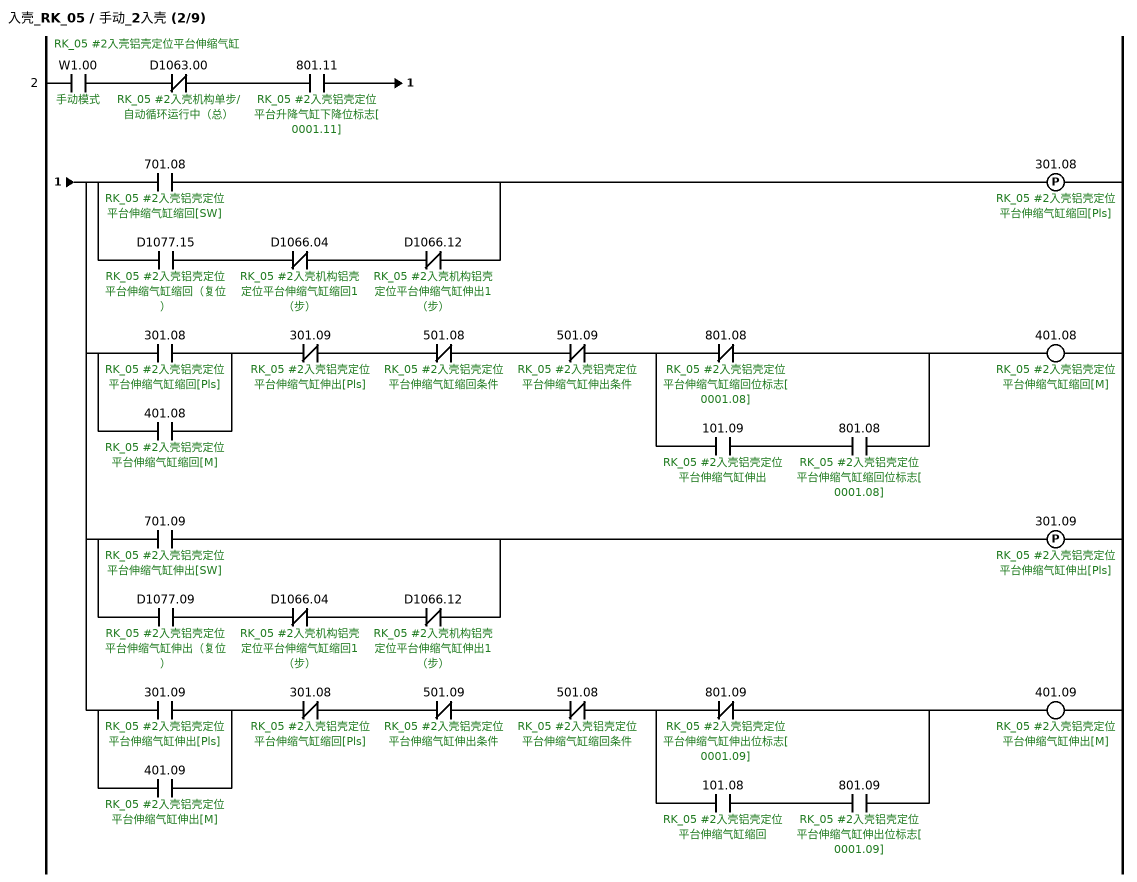
; rung 2: RK_05 #2入壳铝壳定位平台伸缩气缸
LD W1.00  ; 手动模式
ANDNOT D1063.00  ; RK_05 #2入壳机构单步/自动循环运行中（总）
AND 801.11  ; RK_05 #2入壳铝壳定位平台升降气缸下降位标志[0001.11]
OUT TR0
LD 701.08  ; RK_05 #2入壳铝壳定位平台伸缩气缸缩回[SW]
LD D1077.15  ; RK_05 #2入壳铝壳定位平台伸缩气缸缩回（复位）
ANDNOT D1066.04  ; RK_05 #2入壳机构铝壳定位平台伸缩气缸缩回1（步）
ANDNOT D1066.12  ; RK_05 #2入壳机构铝壳定位平台伸缩气缸伸出1（步）
ORLD
ANDLD
DIFU(013) 301.08  ; RK_05 #2入壳铝壳定位平台伸缩气缸缩回[Pls]
LD TR0
LD 301.08  ; RK_05 #2入壳铝壳定位平台伸缩气缸缩回[Pls]
OR 401.08  ; RK_05 #2入壳铝壳定位平台伸缩气缸缩回[M]
ANDLD
ANDNOT 301.09  ; RK_05 #2入壳铝壳定位平台伸缩气缸伸出[Pls]
ANDNOT 501.08  ; RK_05 #2入壳铝壳定位平台伸缩气缸缩回条件
ANDNOT 501.09  ; RK_05 #2入壳铝壳定位平台伸缩气缸伸出条件
LDNOT 801.08  ; RK_05 #2入壳铝壳定位平台伸缩气缸缩回位标志[0001.08]
LD 101.09  ; RK_05 #2入壳铝壳定位平台伸缩气缸伸出
AND 801.08  ; RK_05 #2入壳铝壳定位平台伸缩气缸缩回位标志[0001.08]
ORLD
ANDLD
OUT 401.08  ; RK_05 #2入壳铝壳定位平台伸缩气缸缩回[M]
LD TR0
LD 701.09  ; RK_05 #2入壳铝壳定位平台伸缩气缸伸出[SW]
LD D1077.09  ; RK_05 #2入壳铝壳定位平台伸缩气缸伸出（复位）
ANDNOT D1066.04  ; RK_05 #2入壳机构铝壳定位平台伸缩气缸缩回1（步）
ANDNOT D1066.12  ; RK_05 #2入壳机构铝壳定位平台伸缩气缸伸出1（步）
ORLD
ANDLD
DIFU(013) 301.09  ; RK_05 #2入壳铝壳定位平台伸缩气缸伸出[Pls]
LD TR0
LD 301.09  ; RK_05 #2入壳铝壳定位平台伸缩气缸伸出[Pls]
OR 401.09  ; RK_05 #2入壳铝壳定位平台伸缩气缸伸出[M]
ANDLD
ANDNOT 301.08  ; RK_05 #2入壳铝壳定位平台伸缩气缸缩回[Pls]
ANDNOT 501.09  ; RK_05 #2入壳铝壳定位平台伸缩气缸伸出条件
ANDNOT 501.08  ; RK_05 #2入壳铝壳定位平台伸缩气缸缩回条件
LDNOT 801.09  ; RK_05 #2入壳铝壳定位平台伸缩气缸伸出位标志[0001.09]
LD 101.08  ; RK_05 #2入壳铝壳定位平台伸缩气缸缩回
AND 801.09  ; RK_05 #2入壳铝壳定位平台伸缩气缸伸出位标志[0001.09]
ORLD
ANDLD
OUT 401.09  ; RK_05 #2入壳铝壳定位平台伸缩气缸伸出[M]

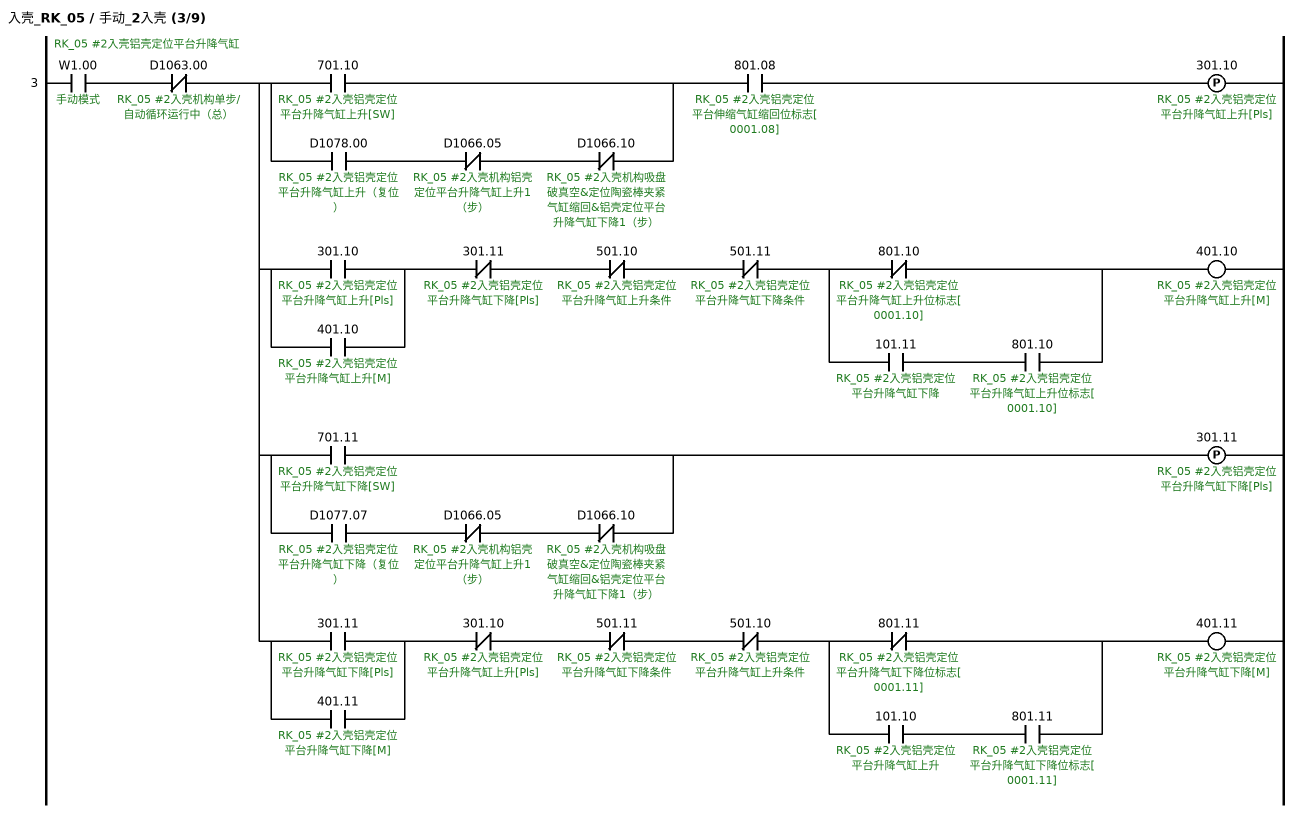
; rung 3: RK_05 #2入壳铝壳定位平台升降气缸
LD W1.00  ; 手动模式
ANDNOT D1063.00  ; RK_05 #2入壳机构单步/自动循环运行中（总）
OUT TR0
LD 701.10  ; RK_05 #2入壳铝壳定位平台升降气缸上升[SW]
LD D1078.00  ; RK_05 #2入壳铝壳定位平台升降气缸上升（复位）
ANDNOT D1066.05  ; RK_05 #2入壳机构铝壳定位平台升降气缸上升1（步）
ANDNOT D1066.10  ; RK_05 #2入壳机构吸盘破真空&定位陶瓷棒夹紧气缸缩回&铝壳定位平台升降气缸下降1（步）
ORLD
ANDLD
AND 801.08  ; RK_05 #2入壳铝壳定位平台伸缩气缸缩回位标志[0001.08]
DIFU(013) 301.10  ; RK_05 #2入壳铝壳定位平台升降气缸上升[Pls]
LD TR0
LD 301.10  ; RK_05 #2入壳铝壳定位平台升降气缸上升[Pls]
OR 401.10  ; RK_05 #2入壳铝壳定位平台升降气缸上升[M]
ANDLD
ANDNOT 301.11  ; RK_05 #2入壳铝壳定位平台升降气缸下降[Pls]
ANDNOT 501.10  ; RK_05 #2入壳铝壳定位平台升降气缸上升条件
ANDNOT 501.11  ; RK_05 #2入壳铝壳定位平台升降气缸下降条件
LDNOT 801.10  ; RK_05 #2入壳铝壳定位平台升降气缸上升位标志[0001.10]
LD 101.11  ; RK_05 #2入壳铝壳定位平台升降气缸下降
AND 801.10  ; RK_05 #2入壳铝壳定位平台升降气缸上升位标志[0001.10]
ORLD
ANDLD
OUT 401.10  ; RK_05 #2入壳铝壳定位平台升降气缸上升[M]
LD TR0
LD 701.11  ; RK_05 #2入壳铝壳定位平台升降气缸下降[SW]
LD D1077.07  ; RK_05 #2入壳铝壳定位平台升降气缸下降（复位）
ANDNOT D1066.05  ; RK_05 #2入壳机构铝壳定位平台升降气缸上升1（步）
ANDNOT D1066.10  ; RK_05 #2入壳机构吸盘破真空&定位陶瓷棒夹紧气缸缩回&铝壳定位平台升降气缸下降1（步）
ORLD
ANDLD
DIFU(013) 301.11  ; RK_05 #2入壳铝壳定位平台升降气缸下降[Pls]
LD TR0
LD 301.11  ; RK_05 #2入壳铝壳定位平台升降气缸下降[Pls]
OR 401.11  ; RK_05 #2入壳铝壳定位平台升降气缸下降[M]
ANDLD
ANDNOT 301.10  ; RK_05 #2入壳铝壳定位平台升降气缸上升[Pls]
ANDNOT 501.11  ; RK_05 #2入壳铝壳定位平台升降气缸下降条件
ANDNOT 501.10  ; RK_05 #2入壳铝壳定位平台升降气缸上升条件
LDNOT 801.11  ; RK_05 #2入壳铝壳定位平台升降气缸下降位标志[0001.11]
LD 101.10  ; RK_05 #2入壳铝壳定位平台升降气缸上升
AND 801.11  ; RK_05 #2入壳铝壳定位平台升降气缸下降位标志[0001.11]
ORLD
ANDLD
OUT 401.11  ; RK_05 #2入壳铝壳定位平台升降气缸下降[M]

